   DATA[168,35] := 250.9933;
   DATA[168,36] := 1.681991;
   DATA[168,37] := 189.6789;
   DATA[168,38] := 0.000128152;
   DATA[168,39] := 1.0;
   DATA[169,0] := 2.625628;
   DATA[169,1] := 525.4767;
   DATA[169,2] := 2.0;
   DATA[169,3] := 2.0;
   DATA[169,4] := 262.0802;
   DATA[169,5] := 8.39163;
   DATA[169,6] := 328.2748;
   DATA[169,7] := 2.445904;
   DATA[169,8] := 2.0;
   DATA[169,9] := 2.0;
   DATA[169,10] := 2.0;
   DATA[169,11] := 19.7964;
   DATA[169,12] := 2.209525;
   DATA[169,13] := 963.2146;
   DATA[169,14] := 1.0;
   DATA[169,15] := 2.0;
   DATA[169,16] := 1.0;
   DATA[169,17] := 1.0;
   DATA[169,18] := 1.0;
   DATA[169,19] := 2.0;
   DATA[169,20] := 148.808;
   DATA[169,21] := 156.1138;
   DATA[169,22] := 1.717489;
   DATA[169,23] := 954.14;
   DATA[169,24] := 2.0;
   DATA[169,25] := 2.0;
   DATA[169,26] := 7.875737;
   DATA[169,27] := 145.1423;
   DATA[169,28] := 264.2271;
   DATA[169,29] := 12.26609;
   DATA[169,30] := 1.726737;
   DATA[169,31] := 1.318816;
   DATA[169,32] := 0.7360369;
   DATA[169,33] := 0.3086186;
   DATA[169,34] := 2.0;
   DATA[169,35] := 250.9933;
   DATA[169,36] := 1.681991;
   DATA[169,37] := 189.6789;
   DATA[169,38] := 0.000128152;
   DATA[169,39] := 1.0;
   DATA[170,0] := 2.624027;
   DATA[170,1] := 525.7122;
   DATA[170,2] := 2.0;
   DATA[170,3] := 2.0;
   DATA[170,4] := 262.0802;
   DATA[170,5] := 8.39163;
   DATA[170,6] := 328.2748;
   DATA[170,7] := 2.444366;
   DATA[170,8] := 2.0;
   DATA[170,9] := 2.0;
   DATA[170,10] := 2.0;
   DATA[170,11] := 19.68756;
   DATA[170,12] := 2.210806;
   DATA[170,13] := 963.1745;
   DATA[170,14] := 1.0;
   DATA[170,15] := 2.0;
   DATA[170,16] := 1.0;
   DATA[170,17] := 1.0;
   DATA[170,18] := 1.0;
   DATA[170,19] := 2.0;
   DATA[170,20] := 148.808;
   DATA[170,21] := 156.1138;
   DATA[170,22] := 1.717489;
   DATA[170,23] := 954.1784;
   DATA[170,24] := 2.0;
   DATA[170,25] := 2.0;
   DATA[170,26] := 7.875737;
   DATA[170,27] := 145.1423;
   DATA[170,28] := 264.2271;
   DATA[170,29] := 12.26609;
   DATA[170,30] := 1.726737;
   DATA[170,31] := 1.322019;
   DATA[170,32] := 0.7360369;
   DATA[170,33] := 0.3084265;
   DATA[170,34] := 2.0;
   DATA[170,35] := 250.9933;
   DATA[170,36] := 1.681991;
   DATA[170,37] := 189.6789;
   DATA[170,38] := 0.000128152;
   DATA[170,39] := 1.0;
   DATA[171,0] := 2.612177;
   DATA[171,1] := 525.8692;
   DATA[171,2] := 2.0;
   DATA[171,3] := 2.0;
   DATA[171,4] := 262.0802;
   DATA[171,5] := 8.39163;
   DATA[171,6] := 328.2748;
   DATA[171,7] := 2.443725;
   DATA[171,8] := 2.0;
   DATA[171,9] := 2.0;
   DATA[171,10] := 2.0;
   DATA[171,11] := 19.68756;
   DATA[171,12] := 2.212728;
   DATA[171,13] := 963.3347;
   DATA[171,14] := 1.0;
   DATA[171,15] := 2.0;
   DATA[171,16] := 1.0;
   DATA[171,17] := 1.0;
   DATA[171,18] := 1.0;
   DATA[171,19] := 2.0;
   DATA[171,20] := 148.808;
   DATA[171,21] := 156.1138;
   DATA[171,22] := 1.717489;
   DATA[171,23] := 954.14;
   DATA[171,24] := 2.0;
   DATA[171,25] := 2.0;
   DATA[171,26] := 7.875737;
   DATA[171,27] := 145.1423;
   DATA[171,28] := 264.2271;
   DATA[171,29] := 12.26609;
   DATA[171,30] := 1.726737;
   DATA[171,31] := 1.322019;
   DATA[171,32] := 0.7353967;
   DATA[171,33] := 0.3074016;
   DATA[171,34] := 2.0;
   DATA[171,35] := 250.9933;
   DATA[171,36] := 1.681991;
   DATA[171,37] := 189.6789;
   DATA[171,38] := 0.000128152;
   DATA[171,39] := 1.0;
   DATA[172,0] := 2.59232;
   DATA[172,1] := 526.1832;
   DATA[172,2] := 2.0;
   DATA[172,3] := 2.0;
   DATA[172,4] := 262.0802;
   DATA[172,5] := 8.396116;
   DATA[172,6] := 328.2748;
   DATA[172,7] := 2.441034;
   DATA[172,8] := 2.0;
   DATA[172,9] := 2.0;
   DATA[172,10] := 2.0;
   DATA[172,11] := 19.68756;
   DATA[172,12] := 2.212728;
   DATA[172,13] := 963.6151;
   DATA[172,14] := 1.0;
   DATA[172,15] := 2.0;
   DATA[172,16] := 1.0;
   DATA[172,17] := 1.0;
   DATA[172,18] := 1.0;
   DATA[172,19] := 2.0;
   DATA[172,20] := 148.808;
   DATA[172,21] := 156.1138;
   DATA[172,22] := 1.717489;
   DATA[172,23] := 954.0246;
   DATA[172,24] := 2.0;
   DATA[172,25] := 2.0;
   DATA[172,26] := 7.875737;
   DATA[172,27] := 145.1423;
   DATA[172,28] := 264.2271;
   DATA[172,29] := 12.26609;
   DATA[172,30] := 1.726737;
   DATA[172,31] := 1.302421;
   DATA[172,32] := 0.7352687;
   DATA[172,33] := 0.3070813;
   DATA[172,34] := 2.0;
   DATA[172,35] := 250.9933;
   DATA[172,36] := 1.681991;
   DATA[172,37] := 189.6789;
   DATA[172,38] := 0.000128152;
   DATA[172,39] := 1.0;
   DATA[173,0] := 2.575665;
   DATA[173,1] := 526.3795;
   DATA[173,2] := 2.0;
   DATA[173,3] := 2.0;
   DATA[173,4] := 262.0802;
   DATA[173,5] := 8.396116;
   DATA[173,6] := 328.2748;
   DATA[173,7] := 2.440778;
   DATA[173,8] := 2.0;
   DATA[173,9] := 2.0;
   DATA[173,10] := 2.0;
   DATA[173,11] := 19.68756;
   DATA[173,12] := 2.212728;
   DATA[173,13] := 963.3748;
   DATA[173,14] := 1.0;
   DATA[173,15] := 2.0;
   DATA[173,16] := 1.0;
   DATA[173,17] := 1.0;
   DATA[173,18] := 1.0;
   DATA[173,19] := 2.0;
   DATA[173,20] := 148.808;
   DATA[173,21] := 156.1138;
   DATA[173,22] := 1.717489;
   DATA[173,23] := 954.1015;
   DATA[173,24] := 2.0;
   DATA[173,25] := 2.0;
   DATA[173,26] := 7.875737;
   DATA[173,27] := 145.1423;
   DATA[173,28] := 264.2271;
   DATA[173,29] := 12.26609;
   DATA[173,30] := 1.725583;
   DATA[173,31] := 1.292046;
   DATA[173,32] := 0.7352687;
   DATA[173,33] := 0.3070813;
   DATA[173,34] := 2.0;
   DATA[173,35] := 250.8812;
   DATA[173,36] := 1.681991;
   DATA[173,37] := 189.6789;
   DATA[173,38] := 0.000128152;
   DATA[173,39] := 1.0;
   DATA[174,0] := 2.554527;
   DATA[174,1] := 526.615;
   DATA[174,2] := 2.0;
   DATA[174,3] := 2.0;
   DATA[174,4] := 262.0802;
   DATA[174,5] := 8.396116;
   DATA[174,6] := 328.2748;
   DATA[174,7] := 2.440778;
   DATA[174,8] := 2.0;
   DATA[174,9] := 2.0;
   DATA[174,10] := 2.0;
   DATA[174,11] := 19.68756;
   DATA[174,12] := 2.211831;
   DATA[174,13] := 963.7353;
   DATA[174,14] := 1.0;
   DATA[174,15] := 2.0;
   DATA[174,16] := 1.0;
   DATA[174,17] := 1.0;
   DATA[174,18] := 1.0;
   DATA[174,19] := 2.0;
   DATA[174,20] := 148.808;
   DATA[174,21] := 156.1138;
   DATA[174,22] := 1.717489;
   DATA[174,23] := 954.5245;
   DATA[174,24] := 2.0;
   DATA[174,25] := 2.0;
   DATA[174,26] := 7.875737;
   DATA[174,27] := 145.1423;
   DATA[174,28] := 264.2271;
   DATA[174,29] := 12.26609;
   DATA[174,30] := 1.725455;
   DATA[174,31] := 1.290893;
   DATA[174,32] := 0.7352687;
   DATA[174,33] := 0.3065048;
   DATA[174,34] := 2.0;
   DATA[174,35] := 250.8812;
   DATA[174,36] := 1.681991;
   DATA[174,37] := 189.6469;
   DATA[174,38] := 0.000128152;
   DATA[174,39] := 1.0;
   DATA[175,0] := 2.535951;
   DATA[175,1] := 526.5757;
   DATA[175,2] := 2.0;
   DATA[175,3] := 2.0;
   DATA[175,4] := 262.0802;
   DATA[175,5] := 8.396116;
   DATA[175,6] := 328.2748;
   DATA[175,7] := 2.441547;
   DATA[175,8] := 2.0;
   DATA[175,9] := 2.0;
   DATA[175,10] := 2.0;
   DATA[175,11] := 19.68756;
   DATA[175,12] := 2.210294;
   DATA[175,13] := 963.7353;
   DATA[175,14] := 1.0;
   DATA[175,15] := 2.0;
   DATA[175,16] := 1.0;
   DATA[175,17] := 1.0;
   DATA[175,18] := 1.0;
   DATA[175,19] := 2.0;
   DATA[175,20] := 148.808;
   DATA[175,21] := 156.1138;
   DATA[175,22] := 1.717489;
   DATA[175,23] := 955.1013;
   DATA[175,24] := 2.0;
   DATA[175,25] := 2.0;
   DATA[175,26] := 7.875737;
   DATA[175,27] := 145.1423;
   DATA[175,28] := 264.2271;
   DATA[175,29] := 12.11228;
   DATA[175,30] := 1.725455;
   DATA[175,31] := 1.285001;
   DATA[175,32] := 0.7352687;
   DATA[175,33] := 0.3065048;
   DATA[175,34] := 2.0;
   DATA[175,35] := 250.8812;
   DATA[175,36] := 1.681991;
   DATA[175,37] := 189.5347;
   DATA[175,38] := 0.000128152;
   DATA[175,39] := 1.0;
   DATA[176,0] := 2.520257;
   DATA[176,1] := 526.6542;
   DATA[176,2] := 2.0;
   DATA[176,3] := 2.0;
   DATA[176,4] := 262.0802;
   DATA[176,5] := 8.396116;
   DATA[176,6] := 328.2748;
   DATA[176,7] := 2.443597;
   DATA[176,8] := 2.0;
   DATA[176,9] := 2.0;
   DATA[176,10] := 2.0;
   DATA[176,11] := 19.68756;
   DATA[176,12] := 2.210166;
   DATA[176,13] := 963.535;
   DATA[176,14] := 1.0;
   DATA[176,15] := 2.0;
   DATA[176,16] := 1.0;
   DATA[176,17] := 1.0;
   DATA[176,18] := 1.0;
   DATA[176,19] := 2.0;
   DATA[176,20] := 148.808;
   DATA[176,21] := 156.0369;
   DATA[176,22] := 1.717489;
   DATA[176,23] := 955.3704;
   DATA[176,24] := 2.0;
   DATA[176,25] := 2.0;
   DATA[176,26] := 7.875737;
   DATA[176,27] := 145.1423;
   DATA[176,28] := 264.2271;
   DATA[176,29] := 12.11228;
   DATA[176,30] := 1.725455;
   DATA[176,31] := 1.272704;
   DATA[176,32] := 0.7352687;
   DATA[176,33] := 0.3065048;
   DATA[176,34] := 2.0;
   DATA[176,35] := 250.8812;
   DATA[176,36] := 1.681991;
   DATA[176,37] := 189.5347;
   DATA[176,38] := 0.000128152;
   DATA[176,39] := 1.0;
   DATA[177,0] := 2.501041;
   DATA[177,1] := 526.8113;
   DATA[177,2] := 2.0;
   DATA[177,3] := 2.0;
   DATA[177,4] := 262.0802;
   DATA[177,5] := 8.396116;
   DATA[177,6] := 328.2748;
   DATA[177,7] := 2.445391;
   DATA[177,8] := 2.0;
   DATA[177,9] := 2.0;
   DATA[177,10] := 2.0;
   DATA[177,11] := 19.71957;
   DATA[177,12] := 2.210934;
   DATA[177,13] := 963.6151;
   DATA[177,14] := 1.0;
   DATA[177,15] := 2.0;
   DATA[177,16] := 1.0;
   DATA[177,17] := 1.0;
   DATA[177,18] := 1.0;
   DATA[177,19] := 2.0;
   DATA[177,20] := 148.808;
   DATA[177,21] := 155.9087;
   DATA[177,22] := 1.717489;
   DATA[177,23] := 955.2935;
   DATA[177,24] := 2.0;
   DATA[177,25] := 2.0;
   DATA[177,26] := 7.875737;
   DATA[177,27] := 145.091;
   DATA[177,28] := 264.2271;
   DATA[177,29] := 12.11228;
   DATA[177,30] := 1.725455;
   DATA[177,31] := 1.272064;
   DATA[177,32] := 0.7352687;
   DATA[177,33] := 0.3065048;
   DATA[177,34] := 2.0;
   DATA[177,35] := 250.8812;
   DATA[177,36] := 1.681991;
   DATA[177,37] := 189.5347;
   DATA[177,38] := 0.000128152;
   DATA[177,39] := 1.0;
   DATA[178,0] := 2.48823;
   DATA[178,1] := 527.2038;
   DATA[178,2] := 2.0;
   DATA[178,3] := 2.0;
   DATA[178,4] := 262.0802;
   DATA[178,5] := 8.396116;
   DATA[178,6] := 328.2748;
   DATA[178,7] := 2.445391;
   DATA[178,8] := 2.0;
   DATA[178,9] := 2.0;
   DATA[178,10] := 2.0;
   DATA[178,11] := 19.74198;
   DATA[178,12] := 2.213368;
   DATA[178,13] := 963.9756;
   DATA[178,14] := 1.0;
   DATA[178,15] := 2.0;
   DATA[178,16] := 1.0;
   DATA[178,17] := 1.0;
   DATA[178,18] := 1.0;
   DATA[178,19] := 2.0;
   DATA[178,20] := 148.808;
   DATA[178,21] := 155.9087;
   DATA[178,22] := 1.717361;
   DATA[178,23] := 956.0626;
   DATA[178,24] := 2.0;
   DATA[178,25] := 2.0;
   DATA[178,26] := 7.875737;
   DATA[178,27] := 145.091;
   DATA[178,28] := 264.2271;
   DATA[178,29] := 12.11228;
   DATA[178,30] := 1.725455;
   DATA[178,31] := 1.273216;
   DATA[178,32] := 0.7352687;
   DATA[178,33] := 0.3084265;
   DATA[178,34] := 2.0;
   DATA[178,35] := 250.8812;
   DATA[178,36] := 1.681991;
   DATA[178,37] := 189.5347;
   DATA[178,38] := 0.000128152;
   DATA[178,39] := 1.0;
   DATA[179,0] := 2.468693;
   DATA[179,1] := 527.1646;
   DATA[179,2] := 2.0;
   DATA[179,3] := 2.0;
   DATA[179,4] := 262.0802;
   DATA[179,5] := 8.396116;
   DATA[179,6] := 328.2748;
   DATA[179,7] := 2.445391;
   DATA[179,8] := 2.0;
   DATA[179,9] := 2.0;
   DATA[179,10] := 2.0;
   DATA[179,11] := 19.74198;
   DATA[179,12] := 2.213368;
   DATA[179,13] := 964.4562;
   DATA[179,14] := 1.0;
   DATA[179,15] := 2.0;
   DATA[179,16] := 1.0;
   DATA[179,17] := 1.0;
   DATA[179,18] := 1.0;
   DATA[179,19] := 2.0;
   DATA[179,20] := 148.808;
   DATA[179,21] := 155.9087;
   DATA[179,22] := 1.716208;
   DATA[179,23] := 956.3317;
   DATA[179,24] := 2.0;
   DATA[179,25] := 2.0;
   DATA[179,26] := 7.875737;
   DATA[179,27] := 144.9116;
   DATA[179,28] := 264.2271;
   DATA[179,29] := 12.11228;
   DATA[179,30] := 1.725455;
   DATA[179,31] := 1.281542;
   DATA[179,32] := 0.7352687;
   DATA[179,33] := 0.3084265;
   DATA[179,34] := 2.0;
   DATA[179,35] := 250.8812;
   DATA[179,36] := 1.681991;
   DATA[179,37] := 189.5668;
   DATA[179,38] := 0.000128152;
   DATA[179,39] := 1.0;
   DATA[180,0] := 2.451078;
   DATA[180,1] := 527.5571;
   DATA[180,2] := 2.0;
   DATA[180,3] := 2.0;
   DATA[180,4] := 262.0802;
   DATA[180,5] := 8.395475;
   DATA[180,6] := 328.2748;
   DATA[180,7] := 2.445391;
   DATA[180,8] := 2.0;
   DATA[180,9] := 2.0;
   DATA[180,10] := 2.0;
   DATA[180,11] := 19.74198;
   DATA[180,12] := 2.213368;
   DATA[180,13] := 964.8568;
   DATA[180,14] := 1.0;
   DATA[180,15] := 2.0;
   DATA[180,16] := 1.0;
   DATA[180,17] := 1.0;
   DATA[180,18] := 1.0;
   DATA[180,19] := 2.0;
   DATA[180,20] := 148.808;
   DATA[180,21] := 155.9856;
   DATA[180,22] := 1.716208;
   DATA[180,23] := 956.4855;
   DATA[180,24] := 2.0;
   DATA[180,25] := 2.0;
   DATA[180,26] := 7.875737;
   DATA[180,27] := 144.9116;
   DATA[180,28] := 264.2271;
   DATA[180,29] := 12.11228;
   DATA[180,30] := 1.726993;
   DATA[180,31] := 1.281542;
   DATA[180,32] := 0.7352687;
   DATA[180,33] := 0.3084265;
   DATA[180,34] := 2.0;
   DATA[180,35] := 250.8812;
   DATA[180,36] := 1.681991;
   DATA[180,37] := 189.759;
   DATA[180,38] := 0.000128152;
   DATA[180,39] := 1.0;
   DATA[181,0] := 2.440188;
   DATA[181,1] := 527.8318;
   DATA[181,2] := 2.0;
   DATA[181,3] := 2.0;
   DATA[181,4] := 262.0802;
   DATA[181,5] := 8.395475;
   DATA[181,6] := 328.2748;
   DATA[181,7] := 2.44411;
   DATA[181,8] := 2.0;
   DATA[181,9] := 2.0;
   DATA[181,10] := 2.0;
   DATA[181,11] := 19.72598;
   DATA[181,12] := 2.213368;
   DATA[181,13] := 965.2573;
   DATA[181,14] := 1.0;
   DATA[181,15] := 2.0;
   DATA[181,16] := 1.0;
   DATA[181,17] := 1.0;
   DATA[181,18] := 1.0;
   DATA[181,19] := 2.0;
   DATA[181,20] := 148.808;
   DATA[181,21] := 156.0625;
   DATA[181,22] := 1.71813;
   DATA[181,23] := 957.2161;
   DATA[181,24] := 2.0;
   DATA[181,25] := 2.0;
   DATA[181,26] := 7.875737;
   DATA[181,27] := 144.9116;
   DATA[181,28] := 264.2271;
   DATA[181,29] := 12.11228;
   DATA[181,30] := 1.726993;
   DATA[181,31] := 1.281542;
   DATA[181,32] := 0.7352687;
   DATA[181,33] := 0.3084265;
   DATA[181,34] := 2.0;
   DATA[181,35] := 250.9933;
   DATA[181,36] := 1.681991;
   DATA[181,37] := 189.759;
   DATA[181,38] := 0.000128152;
   DATA[181,39] := 1.0;
   DATA[182,0] := 2.429619;
   DATA[182,1] := 527.8318;
   DATA[182,2] := 2.0;
   DATA[182,3] := 2.0;
   DATA[182,4] := 262.0802;
   DATA[182,5] := 8.395475;
   DATA[182,6] := 328.2748;
   DATA[182,7] := 2.44411;
   DATA[182,8] := 2.0;
   DATA[182,9] := 2.0;
   DATA[182,10] := 2.0;
   DATA[182,11] := 19.72598;
   DATA[182,12] := 2.214137;
   DATA[182,13] := 965.5778;
   DATA[182,14] := 1.0;
   DATA[182,15] := 2.0;
   DATA[182,16] := 1.0;
   DATA[182,17] := 1.0;
   DATA[182,18] := 1.0;
   DATA[182,19] := 2.0;
   DATA[182,20] := 148.808;
   DATA[182,21] := 156.0625;
   DATA[182,22] := 1.718771;
   DATA[182,23] := 957.0623;
   DATA[182,24] := 2.0;
   DATA[182,25] := 2.0;
   DATA[182,26] := 7.875737;
   DATA[182,27] := 144.9116;
   DATA[182,28] := 264.131;
   DATA[182,29] := 12.11228;
   DATA[182,30] := 1.728659;
   DATA[182,31] := 1.281542;
   DATA[182,32] := 0.7352687;
   DATA[182,33] := 0.3084265;
   DATA[182,34] := 2.0;
   DATA[182,35] := 251.1215;
   DATA[182,36] := 1.681991;
   DATA[182,37] := 189.759;
   DATA[182,38] := 0.000128152;
   DATA[182,39] := 1.0;
   DATA[183,0] := 2.426737;
   DATA[183,1] := 528.3421;
   DATA[183,2] := 2.0;
   DATA[183,3] := 2.0;
   DATA[183,4] := 262.0802;
   DATA[183,5] := 8.395475;
   DATA[183,6] := 328.2748;
   DATA[183,7] := 2.44411;
   DATA[183,8] := 2.0;
   DATA[183,9] := 2.0;
   DATA[183,10] := 2.0;
   DATA[183,11] := 19.72598;
   DATA[183,12] := 2.214137;
   DATA[183,13] := 965.778;
   DATA[183,14] := 1.0;
   DATA[183,15] := 2.0;
   DATA[183,16] := 1.0;
   DATA[183,17] := 1.0;
   DATA[183,18] := 1.0;
   DATA[183,19] := 2.0;
   DATA[183,20] := 148.808;
   DATA[183,21] := 156.0625;
   DATA[183,22] := 1.718771;
   DATA[183,23] := 957.5621;
   DATA[183,24] := 2.0;
   DATA[183,25] := 2.0;
   DATA[183,26] := 7.875737;
   DATA[183,27] := 144.9116;
   DATA[183,28] := 264.131;
   DATA[183,29] := 12.11228;
   DATA[183,30] := 1.728916;
   DATA[183,31] := 1.275138;
   DATA[183,32] := 0.7352687;
   DATA[183,33] := 0.3084265;
   DATA[183,34] := 2.0;
   DATA[183,35] := 251.1215;
   DATA[183,36] := 1.681991;
   DATA[183,37] := 189.759;
   DATA[183,38] := 0.000128152;
   DATA[183,39] := 1.0;
   DATA[184,0] := 2.428018;
   DATA[184,1] := 528.2636;
   DATA[184,2] := 2.0;
   DATA[184,3] := 2.0;
   DATA[184,4] := 262.0802;
   DATA[184,5] := 8.393232;
   DATA[184,6] := 328.2748;
   DATA[184,7] := 2.443469;
   DATA[184,8] := 2.0;
   DATA[184,9] := 2.0;
   DATA[184,10] := 2.0;
   DATA[184,11] := 19.74838;
   DATA[184,12] := 2.211575;
   DATA[184,13] := 965.6178;
   DATA[184,14] := 1.0;
   DATA[184,15] := 2.0;
   DATA[184,16] := 1.0;
   DATA[184,17] := 1.0;
   DATA[184,18] := 1.0;
   DATA[184,19] := 2.0;
   DATA[184,20] := 148.808;
   DATA[184,21] := 156.0625;
   DATA[184,22] := 1.718771;
   DATA[184,23] := 957.6775;
   DATA[184,24] := 2.0;
   DATA[184,25] := 2.0;
   DATA[184,26] := 7.875737;
   DATA[184,27] := 144.9116;
   DATA[184,28] := 264.131;
   DATA[184,29] := 12.11228;
   DATA[184,30] := 1.729172;
   DATA[184,31] := 1.288331;
   DATA[184,32] := 0.7352687;
   DATA[184,33] := 0.3068891;
   DATA[184,34] := 2.0;
   DATA[184,35] := 251.1215;
   DATA[184,36] := 1.681991;
   DATA[184,37] := 189.9032;
   DATA[184,38] := 0.000128152;
   DATA[184,39] := 1.0;
   DATA[185,0] := 2.480863;
   DATA[185,1] := 528.2244;
   DATA[185,2] := 2.0;
   DATA[185,3] := 2.0;
   DATA[185,4] := 262.0802;
   DATA[185,5] := 8.393232;
   DATA[185,6] := 328.2748;
   DATA[185,7] := 2.442188;
   DATA[185,8] := 2.0;
   DATA[185,9] := 2.0;
   DATA[185,10] := 2.0;
   DATA[185,11] := 19.77079;
   DATA[185,12] := 2.210166;
   DATA[185,13] := 965.9382;
   DATA[185,14] := 1.0;
   DATA[185,15] := 2.0;
   DATA[185,16] := 1.0;
   DATA[185,17] := 1.0;
   DATA[185,18] := 1.0;
   DATA[185,19] := 2.0;
   DATA[185,20] := 148.808;
   DATA[185,21] := 156.0625;
   DATA[185,22] := 1.717489;
   DATA[185,23] := 957.7928;
   DATA[185,24] := 2.0;
   DATA[185,25] := 2.0;
   DATA[185,26] := 7.875737;
   DATA[185,27] := 144.7065;
   DATA[185,28] := 264.131;
   DATA[185,29] := 12.11228;
   DATA[185,30] := 1.729172;
   DATA[185,31] := 1.291149;
   DATA[185,32] := 0.7353967;
   DATA[185,33] := 0.3072094;
   DATA[185,34] := 2.0;
   DATA[185,35] := 251.2657;
   DATA[185,36] := 1.681991;
   DATA[185,37] := 189.9032;
   DATA[185,38] := 0.000128152;
   DATA[185,39] := 1.0;
   DATA[186,0] := 2.528264;
   DATA[186,1] := 528.0674;
   DATA[186,2] := 2.0;
   DATA[186,3] := 2.0;
   DATA[186,4] := 262.0802;
   DATA[186,5] := 8.393232;
   DATA[186,6] := 328.2748;
   DATA[186,7] := 2.442188;
   DATA[186,8] := 2.0;
   DATA[186,9] := 2.0;
   DATA[186,10] := 2.0;
   DATA[186,11] := 19.77079;
   DATA[186,12] := 2.210166;
   DATA[186,13] := 965.8582;
   DATA[186,14] := 1.0;
   DATA[186,15] := 2.0;
   DATA[186,16] := 1.0;
   DATA[186,17] := 1.0;
   DATA[186,18] := 1.0;
   DATA[186,19] := 2.0;
   DATA[186,20] := 148.808;
   DATA[186,21] := 156.0625;
   DATA[186,22] := 1.717489;
   DATA[186,23] := 957.8313;
   DATA[186,24] := 2.0;
   DATA[186,25] := 2.0;
   DATA[186,26] := 7.875737;
   DATA[186,27] := 144.7065;
   DATA[186,28] := 264.131;
   DATA[186,29] := 12.11228;
   DATA[186,30] := 1.729172;
   DATA[186,31] := 1.281798;
   DATA[186,32] := 0.7353967;
   DATA[186,33] := 0.3072094;
   DATA[186,34] := 2.0;
   DATA[186,35] := 251.2657;
   DATA[186,36] := 1.681991;
   DATA[186,37] := 189.9032;
   DATA[186,38] := 0.000128152;
   DATA[186,39] := 1.0;
   DATA[187,0] := 2.56958;
   DATA[187,1] := 528.0674;
   DATA[187,2] := 2.0;
   DATA[187,3] := 2.0;
   DATA[187,4] := 262.0802;
   DATA[187,5] := 8.393232;
   DATA[187,6] := 328.2748;
   DATA[187,7] := 2.441034;
   DATA[187,8] := 2.0;
   DATA[187,9] := 2.0;
   DATA[187,10] := 2.0;
   DATA[187,11] := 19.73878;
   DATA[187,12] := 2.210166;
   DATA[187,13] := 965.5778;
   DATA[187,14] := 1.0;
   DATA[187,15] := 2.0;
   DATA[187,16] := 1.0;
   DATA[187,17] := 1.0;
   DATA[187,18] := 1.0;
   DATA[187,19] := 2.0;
   DATA[187,20] := 148.808;
   DATA[187,21] := 156.0625;
   DATA[187,22] := 1.717489;
   DATA[187,23] := 958.2543;
   DATA[187,24] := 2.0;
   DATA[187,25] := 2.0;
   DATA[187,26] := 7.875737;
   DATA[187,27] := 144.7065;
   DATA[187,28] := 264.131;
   DATA[187,29] := 12.11228;
   DATA[187,30] := 1.729172;
   DATA[187,31] := 1.281286;
   DATA[187,32] := 0.7353967;
   DATA[187,33] := 0.3072094;
   DATA[187,34] := 2.0;
   DATA[187,35] := 251.2657;
   DATA[187,36] := 1.681991;
   DATA[187,37] := 189.9032;
   DATA[187,38] := 0.000128152;
   DATA[187,39] := 1.0;
   DATA[188,0] := 2.601287;
   DATA[188,1] := 528.3421;
   DATA[188,2] := 2.0;
   DATA[188,3] := 2.0;
   DATA[188,4] := 262.0802;
   DATA[188,5] := 8.393232;
   DATA[188,6] := 328.2748;
   DATA[188,7] := 2.440521;
   DATA[188,8] := 2.0;
   DATA[188,9] := 2.0;
   DATA[188,10] := 2.0;
   DATA[188,11] := 19.70037;
   DATA[188,12] := 2.212984;
   DATA[188,13] := 965.4576;
   DATA[188,14] := 1.0;
   DATA[188,15] := 2.0;
   DATA[188,16] := 1.0;
   DATA[188,17] := 1.0;
   DATA[188,18] := 1.0;
   DATA[188,19] := 2.0;
   DATA[188,20] := 148.808;
   DATA[188,21] := 156.0625;
   DATA[188,22] := 1.717489;
   DATA[188,23] := 958.3312;
   DATA[188,24] := 2.0;
   DATA[188,25] := 2.0;
   DATA[188,26] := 7.876378;
   DATA[188,27] := 144.7065;
   DATA[188,28] := 264.131;
   DATA[188,29] := 12.11228;
   DATA[188,30] := 1.729172;
   DATA[188,31] := 1.273216;
   DATA[188,32] := 0.7353967;
   DATA[188,33] := 0.3072094;
   DATA[188,34] := 2.0;
   DATA[188,35] := 251.2657;
   DATA[188,36] := 1.681991;
   DATA[188,37] := 189.9032;
   DATA[188,38] := 0.000128152;
   DATA[188,39] := 1.0;
   DATA[189,0] := 2.644525;
   DATA[189,1] := 528.4207;
   DATA[189,2] := 2.0;
   DATA[189,3] := 2.0;
   DATA[189,4] := 262.0802;
   DATA[189,5] := 8.391951;
   DATA[189,6] := 328.2748;
   DATA[189,7] := 2.440521;
   DATA[189,8] := 2.0;
   DATA[189,9] := 2.0;
   DATA[189,10] := 2.0;
   DATA[189,11] := 19.65875;
   DATA[189,12] := 2.212984;
   DATA[189,13] := 965.3375;
   DATA[189,14] := 1.0;
   DATA[189,15] := 2.0;
   DATA[189,16] := 1.0;
   DATA[189,17] := 1.0;
   DATA[189,18] := 1.0;
   DATA[189,19] := 2.0;
   DATA[189,20] := 148.808;
   DATA[189,21] := 156.0625;
   DATA[189,22] := 1.717489;
   DATA[189,23] := 958.5234;
   DATA[189,24] := 2.0;
   DATA[189,25] := 2.0;
   DATA[189,26] := 7.878621;
   DATA[189,27] := 144.7065;
   DATA[189,28] := 264.131;
   DATA[189,29] := 12.26609;
   DATA[189,30] := 1.729172;
   DATA[189,31] := 1.271935;
   DATA[189,32] := 0.7353967;
   DATA[189,33] := 0.3072094;
   DATA[189,34] := 2.0;
   DATA[189,35] := 251.2657;
   DATA[189,36] := 1.681991;
   DATA[189,37] := 189.9032;
   DATA[189,38] := 0.000128152;
   DATA[189,39] := 1.0;
   DATA[190,0] := 2.665663;
   DATA[190,1] := 528.1851;
   DATA[190,2] := 2.0;
   DATA[190,3] := 2.0;
   DATA[190,4] := 262.0802;
   DATA[190,5] := 8.391951;
   DATA[190,6] := 328.2748;
   DATA[190,7] := 2.440521;
   DATA[190,8] := 2.0;
   DATA[190,9] := 2.0;
   DATA[190,10] := 2.0;
   DATA[190,11] := 19.64274;
   DATA[190,12] := 2.212984;
   DATA[190,13] := 965.3375;
   DATA[190,14] := 1.0;
   DATA[190,15] := 2.0;
   DATA[190,16] := 1.0;
   DATA[190,17] := 1.0;
   DATA[190,18] := 1.0;
   DATA[190,19] := 2.0;
   DATA[190,20] := 148.808;
   DATA[190,21] := 156.0625;
   DATA[190,22] := 1.717489;
   DATA[190,23] := 959.0618;
   DATA[190,24] := 2.0;
   DATA[190,25] := 2.0;
   DATA[190,26] := 7.878621;
   DATA[190,27] := 144.7065;
   DATA[190,28] := 264.131;
   DATA[190,29] := 12.26609;
   DATA[190,30] := 1.729172;
   DATA[190,31] := 1.271935;
   DATA[190,32] := 0.7353967;
   DATA[190,33] := 0.306761;
   DATA[190,34] := 2.0;
   DATA[190,35] := 251.1055;
   DATA[190,36] := 1.681991;
   DATA[190,37] := 189.9032;
   DATA[190,38] := 0.000128152;
   DATA[190,39] := 1.0;
   DATA[191,0] := 2.670788;
   DATA[191,1] := 527.8711;
   DATA[191,2] := 2.0;
   DATA[191,3] := 2.0;
   DATA[191,4] := 262.0802;
   DATA[191,5] := 8.391951;
   DATA[191,6] := 328.2748;
   DATA[191,7] := 2.440521;
   DATA[191,8] := 2.0;
   DATA[191,9] := 2.0;
   DATA[191,10] := 2.0;
   DATA[191,11] := 19.64274;
   DATA[191,12] := 2.212984;
   DATA[191,13] := 965.3775;
   DATA[191,14] := 1.0;
   DATA[191,15] := 2.0;
   DATA[191,16] := 1.0;
   DATA[191,17] := 1.0;
   DATA[191,18] := 1.0;
   DATA[191,19] := 2.0;
   DATA[191,20] := 148.808;
   DATA[191,21] := 156.0625;
   DATA[191,22] := 1.717489;
   DATA[191,23] := 958.9849;
   DATA[191,24] := 2.0;
   DATA[191,25] := 2.0;
   DATA[191,26] := 7.878621;
   DATA[191,27] := 144.7065;
   DATA[191,28] := 264.131;
   DATA[191,29] := 12.26609;
   DATA[191,30] := 1.729172;
   DATA[191,31] := 1.281542;
   DATA[191,32] := 0.7353967;
   DATA[191,33] := 0.3065048;
   DATA[191,34] := 2.0;
   DATA[191,35] := 251.1055;
   DATA[191,36] := 1.681991;
   DATA[191,37] := 189.9032;
   DATA[191,38] := 0.000128152;
   DATA[191,39] := 1.0;
   DATA[192,0] := 2.656055;
   DATA[192,1] := 528.1459;
   DATA[192,2] := 2.0;
   DATA[192,3] := 2.0;
   DATA[192,4] := 262.0802;
   DATA[192,5] := 8.391951;
   DATA[192,6] := 328.2748;
   DATA[192,7] := 2.440521;
   DATA[192,8] := 2.0;
   DATA[192,9] := 2.0;
   DATA[192,10] := 2.0;
   DATA[192,11] := 19.64274;
   DATA[192,12] := 2.213624;
   DATA[192,13] := 965.1772;
   DATA[192,14] := 1.0;
   DATA[192,15] := 2.0;
   DATA[192,16] := 1.0;
   DATA[192,17] := 1.0;
   DATA[192,18] := 1.0;
   DATA[192,19] := 2.0;
   DATA[192,20] := 148.808;
   DATA[192,21] := 156.0625;
   DATA[192,22] := 1.717489;
   DATA[192,23] := 958.9464;
   DATA[192,24] := 2.0;
   DATA[192,25] := 2.0;
   DATA[192,26] := 7.877019;
   DATA[192,27] := 144.7065;
   DATA[192,28] := 264.131;
   DATA[192,29] := 12.26609;
   DATA[192,30] := 1.729172;
   DATA[192,31] := 1.298578;
   DATA[192,32] := 0.7353967;
   DATA[192,33] := 0.3065048;
   DATA[192,34] := 2.0;
   DATA[192,35] := 251.1055;
   DATA[192,36] := 1.681991;
   DATA[192,37] := 189.9032;
   DATA[192,38] := 0.000128152;
   DATA[192,39] := 1.0;
   DATA[193,0] := 2.633315;
   DATA[193,1] := 527.4001;
   DATA[193,2] := 2.0;
   DATA[193,3] := 2.0;
   DATA[193,4] := 262.0802;
   DATA[193,5] := 8.391951;
   DATA[193,6] := 328.2748;
   DATA[193,7] := 2.442828;
   DATA[193,8] := 2.0;
   DATA[193,9] := 2.0;
   DATA[193,10] := 2.0;
   DATA[193,11] := 19.64274;
   DATA[193,12] := 2.213624;
   DATA[193,13] := 965.1772;
   DATA[193,14] := 1.0;
   DATA[193,15] := 2.0;
   DATA[193,16] := 1.0;
   DATA[193,17] := 1.0;
   DATA[193,18] := 1.0;
   DATA[193,19] := 2.0;
   DATA[193,20] := 148.808;
   DATA[193,21] := 156.0625;
   DATA[193,22] := 1.717489;
   DATA[193,23] := 958.9849;
   DATA[193,24] := 2.0;
   DATA[193,25] := 2.0;
   DATA[193,26] := 7.876378;
   DATA[193,27] := 144.7065;
   DATA[193,28] := 264.131;
   DATA[193,29] := 12.26609;
   DATA[193,30] := 1.729172;
   DATA[193,31] := 1.302037;
   DATA[193,32] := 0.7353967;
   DATA[193,33] := 0.3065048;
   DATA[193,34] := 2.0;
   DATA[193,35] := 251.1055;
   DATA[193,36] := 1.681991;
   DATA[193,37] := 189.9032;
   DATA[193,38] := 0.000128152;
   DATA[193,39] := 1.0;
   DATA[194,0] := 2.624027;
   DATA[194,1] := 527.1646;
   DATA[194,2] := 2.0;
   DATA[194,3] := 2.0;
   DATA[194,4] := 262.0802;
   DATA[194,5] := 8.391951;
   DATA[194,6] := 328.2748;
   DATA[194,7] := 2.442956;
   DATA[194,8] := 2.0;
   DATA[194,9] := 2.0;
   DATA[194,10] := 2.0;
   DATA[194,11] := 19.64274;
   DATA[194,12] := 2.213624;
   DATA[194,13] := 964.9369;
   DATA[194,14] := 1.0;
   DATA[194,15] := 2.0;
   DATA[194,16] := 1.0;
   DATA[194,17] := 1.0;
   DATA[194,18] := 1.0;
   DATA[194,19] := 2.0;
   DATA[194,20] := 148.808;
   DATA[194,21] := 156.0625;
   DATA[194,22] := 1.717489;
   DATA[194,23] := 958.9464;
   DATA[194,24] := 2.0;
   DATA[194,25] := 2.0;
   DATA[194,26] := 7.875737;
   DATA[194,27] := 144.7065;
   DATA[194,28] := 264.131;
   DATA[194,29] := 12.26609;
   DATA[194,30] := 1.728531;
   DATA[194,31] := 1.302293;
   DATA[194,32] := 0.7353967;
   DATA[194,33] := 0.3065048;
   DATA[194,34] := 2.0;
   DATA[194,35] := 251.1055;
   DATA[194,36] := 1.681991;
   DATA[194,37] := 189.9032;
   DATA[194,38] := 0.000128152;
   DATA[194,39] := 1.0;
   DATA[195,0] := 2.623387;
   DATA[195,1] := 527.4001;
   DATA[195,2] := 2.0;
   DATA[195,3] := 2.0;
   DATA[195,4] := 262.0802;
   DATA[195,5] := 8.391951;
   DATA[195,6] := 328.2748;
   DATA[195,7] := 2.44616;
   DATA[195,8] := 2.0;
   DATA[195,9] := 2.0;
   DATA[195,10] := 2.0;
   DATA[195,11] := 19.64274;
   DATA[195,12] := 2.213624;
   DATA[195,13] := 965.0571;
   DATA[195,14] := 1.0;
   DATA[195,15] := 2.0;
   DATA[195,16] := 1.0;
   DATA[195,17] := 1.0;
   DATA[195,18] := 1.0;
   DATA[195,19] := 2.0;
   DATA[195,20] := 148.808;
   DATA[195,21] := 156.0625;
   DATA[195,22] := 1.717489;
   DATA[195,23] := 958.9464;
   DATA[195,24] := 2.0;
   DATA[195,25] := 2.0;
   DATA[195,26] := 7.875737;
   DATA[195,27] := 144.7578;
   DATA[195,28] := 264.131;
   DATA[195,29] := 12.26609;
   DATA[195,30] := 1.72725;
   DATA[195,31] := 1.29307;
   DATA[195,32] := 0.7353967;
   DATA[195,33] := 0.3065048;
   DATA[195,34] := 2.0;
   DATA[195,35] := 251.1055;
   DATA[195,36] := 1.681991;
   DATA[195,37] := 189.8071;
   DATA[195,38] := 0.000128152;
   DATA[195,39] := 1.0;
   DATA[196,0] := 2.617942;
   DATA[196,1] := 527.4786;
   DATA[196,2] := 2.0;
   DATA[196,3] := 2.0;
   DATA[196,4] := 262.0802;
   DATA[196,5] := 8.391951;
   DATA[196,6] := 328.2748;
   DATA[196,7] := 2.44616;
   DATA[196,8] := 2.0;
   DATA[196,9] := 2.0;
   DATA[196,10] := 2.0;
   DATA[196,11] := 19.65875;
   DATA[196,12] := 2.213624;
   DATA[196,13] := 965.1772;
   DATA[196,14] := 1.0;
   DATA[196,15] := 2.0;
   DATA[196,16] := 1.0;
   DATA[196,17] := 1.0;
   DATA[196,18] := 1.0;
   DATA[196,19] := 2.0;
   DATA[196,20] := 148.808;
   DATA[196,21] := 156.0625;
   DATA[196,22] := 1.714029;
   DATA[196,23] := 959.1771;
   DATA[196,24] := 2.0;
   DATA[196,25] := 2.0;
   DATA[196,26] := 7.875737;
   DATA[196,27] := 144.7578;
   DATA[196,28] := 264.131;
   DATA[196,29] := 12.26609;
   DATA[196,30] := 1.726737;
   DATA[196,31] := 1.273345;
   DATA[196,32] := 0.7353967;
   DATA[196,33] := 0.3065048;
   DATA[196,34] := 2.0;
   DATA[196,35] := 250.9773;
   DATA[196,36] := 1.826162;
   DATA[196,37] := 189.6789;
   DATA[196,38] := 0.000128152;
   DATA[196,39] := 1.0;
   DATA[197,0] := 2.596163;
   DATA[197,1] := 527.2038;
   DATA[197,2] := 2.0;
   DATA[197,3] := 2.0;
   DATA[197,4] := 262.0802;
   DATA[197,5] := 8.391951;
   DATA[197,6] := 328.2748;
   DATA[197,7] := 2.443982;
   DATA[197,8] := 2.0;
   DATA[197,9] := 2.0;
   DATA[197,10] := 2.0;
   DATA[197,11] := 19.67155;
   DATA[197,12] := 2.213624;
   DATA[197,13] := 964.9369;
   DATA[197,14] := 1.0;
   DATA[197,15] := 2.0;
   DATA[197,16] := 1.0;
   DATA[197,17] := 1.0;
   DATA[197,18] := 1.0;
   DATA[197,19] := 2.0;
   DATA[197,20] := 148.808;
   DATA[197,21] := 156.0625;
   DATA[197,22] := 1.713389;
   DATA[197,23] := 959.1771;
   DATA[197,24] := 2.0;
   DATA[197,25] := 2.0;
   DATA[197,26] := 7.875737;
   DATA[197,27] := 144.7578;
   DATA[197,28] := 264.131;
   DATA[197,29] := 12.26609;
   DATA[197,30] := 1.726737;
   DATA[197,31] := 1.275778;
   DATA[197,32] := 0.7353967;
   DATA[197,33] := 0.3065048;
   DATA[197,34] := 2.0;
   DATA[197,35] := 250.8972;
   DATA[197,36] := 1.826162;
   DATA[197,37] := 189.6148;
   DATA[197,38] := 0.000128152;
   DATA[197,39] := 1.0;
   DATA[198,0] := 2.578548;
   DATA[198,1] := 527.3608;
   DATA[198,2] := 2.0;
   DATA[198,3] := 2.0;
   DATA[198,4] := 262.0802;
   DATA[198,5] := 8.391951;
   DATA[198,6] := 328.2748;
   DATA[198,7] := 2.443085;
   DATA[198,8] := 2.0;
   DATA[198,9] := 2.0;
   DATA[198,10] := 2.0;
   DATA[198,11] := 19.67796;
   DATA[198,12] := 2.213624;
   DATA[198,13] := 964.8167;
   DATA[198,14] := 1.0;
   DATA[198,15] := 2.0;
   DATA[198,16] := 1.0;
   DATA[198,17] := 1.0;
   DATA[198,18] := 1.0;
   DATA[198,19] := 2.0;
   DATA[198,20] := 148.808;
   DATA[198,21] := 156.0625;
   DATA[198,22] := 1.71262;
   DATA[198,23] := 959.3309;
   DATA[198,24] := 2.0;
   DATA[198,25] := 2.0;
   DATA[198,26] := 7.875737;
   DATA[198,27] := 144.7578;
   DATA[198,28] := 264.131;
   DATA[198,29] := 12.26609;
   DATA[198,30] := 1.726737;
   DATA[198,31] := 1.289996;
   DATA[198,32] := 0.7353967;
   DATA[198,33] := 0.3081703;
   DATA[198,34] := 2.0;
   DATA[198,35] := 250.8011;
   DATA[198,36] := 1.649953;
   DATA[198,37] := 189.5187;
   DATA[198,38] := 0.000128152;
   DATA[198,39] := 1.0;
   DATA[199,0] := 2.561573;
   DATA[199,1] := 527.1646;
   DATA[199,2] := 2.0;
   DATA[199,3] := 2.0;
   DATA[199,4] := 262.0802;
   DATA[199,5] := 8.391951;
   DATA[199,6] := 328.2748;
   DATA[199,7] := 2.442828;
   DATA[199,8] := 2.0;
   DATA[199,9] := 2.0;
   DATA[199,10] := 2.0;
   DATA[199,11] := 19.67796;
   DATA[199,12] := 2.213624;
   DATA[199,13] := 964.7767;
   DATA[199,14] := 1.0;
   DATA[199,15] := 2.0;
   DATA[199,16] := 1.0;
   DATA[199,17] := 1.0;
   DATA[199,18] := 1.0;
   DATA[199,19] := 2.0;
   DATA[199,20] := 148.808;
   DATA[199,21] := 156.0625;
   DATA[199,22] := 1.71262;
   DATA[199,23] := 959.2156;
   DATA[199,24] := 2.0;
   DATA[199,25] := 2.0;
   DATA[199,26] := 7.875737;
   DATA[199,27] := 144.7578;
   DATA[199,28] := 264.131;
   DATA[199,29] := 12.15073;
   DATA[199,30] := 1.725455;
   DATA[199,31] := 1.30114;
   DATA[199,32] := 0.7353967;
   DATA[199,33] := 0.3083624;
   DATA[199,34] := 2.0;
   DATA[199,35] := 250.785;
   DATA[199,36] := 1.649953;
   DATA[199,37] := 189.5187;
   DATA[199,38] := 0.000128152;
   DATA[199,39] := 1.0;
   DATA[200,0] := 2.54652;
   DATA[200,1] := 526.8898;
   DATA[200,2] := 2.0;
   DATA[200,3] := 2.0;
   DATA[200,4] := 262.0802;
   DATA[200,5] := 8.391951;
   DATA[200,6] := 328.2748;
   DATA[200,7] := 2.441547;
   DATA[200,8] := 2.0;
   DATA[200,9] := 2.0;
   DATA[200,10] := 2.0;
   DATA[200,11] := 19.67796;
   DATA[200,12] := 2.214906;
   DATA[200,13] := 964.9369;
   DATA[200,14] := 1.0;
   DATA[200,15] := 2.0;
   DATA[200,16] := 1.0;
   DATA[200,17] := 1.0;
   DATA[200,18] := 1.0;
   DATA[200,19] := 2.0;
   DATA[200,20] := 148.808;
   DATA[200,21] := 155.9087;
   DATA[200,22] := 1.71262;
   DATA[200,23] := 959.254;
   DATA[200,24] := 2.0;
   DATA[200,25] := 2.0;
   DATA[200,26] := 7.875737;
   DATA[200,27] := 144.7578;
   DATA[200,28] := 264.131;
   DATA[200,29] := 12.03538;
   DATA[200,30] := 1.72507;
   DATA[200,31] := 1.30178;
   DATA[200,32] := 0.7353967;
   DATA[200,33] := 0.3083624;
   DATA[200,34] := 2.0;
   DATA[200,35] := 250.785;
   DATA[200,36] := 1.649953;
   DATA[200,37] := 189.5187;
   DATA[200,38] := 0.000128152;
   DATA[200,39] := 1.0;
   DATA[201,0] := 2.52282;
   DATA[201,1] := 526.772;
   DATA[201,2] := 2.0;
   DATA[201,3] := 2.0;
   DATA[201,4] := 262.0802;
   DATA[201,5] := 8.391951;
   DATA[201,6] := 328.2748;
   DATA[201,7] := 2.440137;
   DATA[201,8] := 2.0;
   DATA[201,9] := 2.0;
   DATA[201,10] := 2.0;
   DATA[201,11] := 19.67796;
   DATA[201,12] := 2.214906;
   DATA[201,13] := 965.0571;
   DATA[201,14] := 1.0;
   DATA[201,15] := 2.0;
   DATA[201,16] := 1.0;
   DATA[201,17] := 1.0;
   DATA[201,18] := 1.0;
   DATA[201,19] := 2.0;
   DATA[201,20] := 148.808;
   DATA[201,21] := 155.9087;
   DATA[201,22] := 1.71262;
   DATA[201,23] := 959.3309;
   DATA[201,24] := 2.0;
   DATA[201,25] := 2.0;
   DATA[201,26] := 7.875737;
   DATA[201,27] := 144.7578;
   DATA[201,28] := 264.131;
   DATA[201,29] := 12.03538;
   DATA[201,30] := 1.724814;
   DATA[201,31] := 1.311259;
   DATA[201,32] := 0.7353967;
   DATA[201,33] := 0.3083624;
   DATA[201,34] := 2.0;
   DATA[201,35] := 250.785;
   DATA[201,36] := 1.778105;
   DATA[201,37] := 189.5187;
   DATA[201,38] := 0.000128152;
   DATA[201,39] := 1.0;
   DATA[202,0] := 2.503283;
   DATA[202,1] := 526.4973;
   DATA[202,2] := 2.0;
   DATA[202,3] := 2.0;
   DATA[202,4] := 262.0802;
   DATA[202,5] := 8.394835;
   DATA[202,6] := 328.2748;
   DATA[202,7] := 2.440137;
   DATA[202,8] := 2.0;
   DATA[202,9] := 2.0;
   DATA[202,10] := 2.0;
   DATA[202,11] := 19.67796;
   DATA[202,12] := 2.212343;
   DATA[202,13] := 965.0571;
   DATA[202,14] := 1.0;
   DATA[202,15] := 2.0;
   DATA[202,16] := 1.0;
   DATA[202,17] := 1.0;
   DATA[202,18] := 1.0;
   DATA[202,19] := 2.0;
   DATA[202,20] := 148.808;
   DATA[202,21] := 155.9087;
   DATA[202,22] := 1.714798;
   DATA[202,23] := 959.2156;
   DATA[202,24] := 2.0;
   DATA[202,25] := 2.0;
   DATA[202,26] := 7.875737;
   DATA[202,27] := 144.7578;
   DATA[202,28] := 264.131;
   DATA[202,29] := 12.03538;
   DATA[202,30] := 1.724814;
   DATA[202,31] := 1.305623;
   DATA[202,32] := 0.7353967;
   DATA[202,33] := 0.3083624;
   DATA[202,34] := 2.0;
   DATA[202,35] := 250.785;
   DATA[202,36] := 1.778105;
   DATA[202,37] := 189.5187;
   DATA[202,38] := 0.000128152;
   DATA[202,39] := 1.0;
   DATA[203,0] := 2.485027;
   DATA[203,1] := 526.301;
   DATA[203,2] := 2.0;
   DATA[203,3] := 2.0;
   DATA[203,4] := 262.0802;
   DATA[203,5] := 8.394835;
   DATA[203,6] := 328.2748;
   DATA[203,7] := 2.440137;
   DATA[203,8] := 2.0;
   DATA[203,9] := 2.0;
   DATA[203,10] := 2.0;
   DATA[203,11] := 19.70037;
   DATA[203,12] := 2.212343;
   DATA[203,13] := 965.3775;
   DATA[203,14] := 1.0;
   DATA[203,15] := 2.0;
   DATA[203,16] := 1.0;
   DATA[203,17] := 1.0;
   DATA[203,18] := 1.0;
   DATA[203,19] := 2.0;
   DATA[203,20] := 148.808;
   DATA[203,21] := 155.9087;
   DATA[203,22] := 1.717233;
   DATA[203,23] := 959.2156;
   DATA[203,24] := 2.0;
   DATA[203,25] := 2.0;
   DATA[203,26] := 7.875737;
   DATA[203,27] := 144.7578;
   DATA[203,28] := 264.131;
   DATA[203,29] := 12.03538;
   DATA[203,30] := 1.726096;
   DATA[203,31] := 1.292558;
   DATA[203,32] := 0.7353967;
   DATA[203,33] := 0.3083624;
   DATA[203,34] := 2.0;
   DATA[203,35] := 250.785;
   DATA[203,36] := 1.778105;
   DATA[203,37] := 189.5187;
   DATA[203,38] := 0.000128152;
   DATA[203,39] := 1.0;
   DATA[204,0] := 2.467092;
   DATA[204,1] := 526.0262;
   DATA[204,2] := 2.0;
   DATA[204,3] := 2.0;
   DATA[204,4] := 262.0802;
   DATA[204,5] := 8.394835;
   DATA[204,6] := 328.2748;
   DATA[204,7] := 2.441547;
   DATA[204,8] := 2.0;
   DATA[204,9] := 2.0;
   DATA[204,10] := 2.0;
   DATA[204,11] := 19.73238;
   DATA[204,12] := 2.209525;
   DATA[204,13] := 965.4576;
   DATA[204,14] := 1.0;
   DATA[204,15] := 2.0;
   DATA[204,16] := 1.0;
   DATA[204,17] := 1.0;
   DATA[204,18] := 1.0;
   DATA[204,19] := 2.0;
   DATA[204,20] := 148.808;
   DATA[204,21] := 155.9087;
   DATA[204,22] := 1.717489;
   DATA[204,23] := 958.8695;
   DATA[204,24] := 2.0;
   DATA[204,25] := 2.0;
   DATA[204,26] := 7.875737;
   DATA[204,27] := 144.7578;
   DATA[204,28] := 264.131;
   DATA[204,29] := 12.03538;
   DATA[204,30] := 1.726096;
   DATA[204,31] := 1.292174;
   DATA[204,32] := 0.7353967;
   DATA[204,33] := 0.3083624;
   DATA[204,34] := 2.0;
   DATA[204,35] := 250.8812;
   DATA[204,36] := 1.778105;
   DATA[204,37] := 189.5187;
   DATA[204,38] := 0.000128152;
   DATA[204,39] := 1.0;
   DATA[205,0] := 2.452679;
   DATA[205,1] := 526.0262;
   DATA[205,2] := 2.0;
   DATA[205,3] := 2.0;
   DATA[205,4] := 262.0802;
   DATA[205,5] := 8.394835;
   DATA[205,6] := 328.2748;
   DATA[205,7] := 2.441547;
   DATA[205,8] := 2.0;
   DATA[205,9] := 2.0;
   DATA[205,10] := 2.0;
   DATA[205,11] := 19.73238;
   DATA[205,12] := 2.209269;
   DATA[205,13] := 965.5778;
   DATA[205,14] := 1.0;
   DATA[205,15] := 2.0;
   DATA[205,16] := 1.0;
   DATA[205,17] := 1.0;
   DATA[205,18] := 1.0;
   DATA[205,19] := 2.0;
   DATA[205,20] := 148.808;
   DATA[205,21] := 155.9087;
   DATA[205,22] := 1.717489;
   DATA[205,23] := 958.8311;
   DATA[205,24] := 2.0;
   DATA[205,25] := 2.0;
   DATA[205,26] := 7.875737;
   DATA[205,27] := 144.7578;
   DATA[205,28] := 264.131;
   DATA[205,29] := 12.03538;
   DATA[205,30] := 1.726737;
   DATA[205,31] := 1.282311;
   DATA[205,32] := 0.7353967;
   DATA[205,33] := 0.3083624;
   DATA[205,34] := 2.0;
   DATA[205,35] := 250.9132;
   DATA[205,36] := 1.69801;
   DATA[205,37] := 189.6629;
   DATA[205,38] := 0.000128152;
   DATA[205,39] := 1.0;
   DATA[206,0] := 2.436345;
   DATA[206,1] := 525.83;
   DATA[206,2] := 2.0;
   DATA[206,3] := 2.0;
   DATA[206,4] := 262.0802;
   DATA[206,5] := 8.394835;
   DATA[206,6] := 328.2748;
   DATA[206,7] := 2.4427;
   DATA[206,8] := 2.0;
   DATA[206,9] := 2.0;
   DATA[206,10] := 2.0;
   DATA[206,11] := 19.67476;
   DATA[206,12] := 2.208372;
   DATA[206,13] := 965.6178;
   DATA[206,14] := 1.0;
   DATA[206,15] := 2.0;
   DATA[206,16] := 1.0;
   DATA[206,17] := 1.0;
   DATA[206,18] := 1.0;
   DATA[206,19] := 2.0;
   DATA[206,20] := 148.808;
   DATA[206,21] := 155.9087;
   DATA[206,22] := 1.717489;
   DATA[206,23] := 958.6388;
   DATA[206,24] := 2.0;
   DATA[206,25] := 2.0;
   DATA[206,26] := 7.875737;
   DATA[206,27] := 144.7578;
   DATA[206,28] := 264.131;
   DATA[206,29] := 12.03538;
   DATA[206,30] := 1.726737;
   DATA[206,31] := 1.281798;
   DATA[206,32] := 0.7353967;
   DATA[206,33] := 0.3083624;
   DATA[206,34] := 2.0;
   DATA[206,35] := 250.9132;
   DATA[206,36] := 1.69801;
   DATA[206,37] := 189.759;
   DATA[206,38] := 0.000128152;
   DATA[206,39] := 1.0;
   DATA[207,0] := 2.428979;
   DATA[207,1] := 525.4767;
   DATA[207,2] := 2.0;
   DATA[207,3] := 2.0;
   DATA[207,4] := 262.0802;
   DATA[207,5] := 8.394835;
   DATA[207,6] := 328.2748;
   DATA[207,7] := 2.443469;
   DATA[207,8] := 2.0;
   DATA[207,9] := 2.0;
   DATA[207,10] := 2.0;
   DATA[207,11] := 19.64594;
   DATA[207,12] := 2.207731;
   DATA[207,13] := 966.1385;
   DATA[207,14] := 1.0;
   DATA[207,15] := 2.0;
   DATA[207,16] := 1.0;
   DATA[207,17] := 1.0;
   DATA[207,18] := 1.0;
   DATA[207,19] := 2.0;
   DATA[207,20] := 148.808;
   DATA[207,21] := 155.9087;
   DATA[207,22] := 1.716464;
   DATA[207,23] := 958.6388;
   DATA[207,24] := 2.0;
   DATA[207,25] := 2.0;
   DATA[207,26] := 7.875737;
   DATA[207,27] := 144.7578;
   DATA[207,28] := 264.131;
   DATA[207,29] := 12.03538;
   DATA[207,30] := 1.726737;
   DATA[207,31] := 1.281542;
   DATA[207,32] := 0.7353967;
   DATA[207,33] := 0.3083624;
   DATA[207,34] := 2.0;
   DATA[207,35] := 250.9132;
   DATA[207,36] := 1.69801;
   DATA[207,37] := 189.759;
   DATA[207,38] := 0.000128152;
   DATA[207,39] := 1.0;
   DATA[208,0] := 2.423534;
   DATA[208,1] := 525.5944;
   DATA[208,2] := 2.0;
   DATA[208,3] := 2.0;
   DATA[208,4] := 262.0802;
   DATA[208,5] := 8.394835;
   DATA[208,6] := 328.2748;
   DATA[208,7] := 2.443725;
   DATA[208,8] := 2.0;
   DATA[208,9] := 2.0;
   DATA[208,10] := 2.0;
   DATA[208,11] := 19.64594;
   DATA[208,12] := 2.207731;
   DATA[208,13] := 966.3788;
   DATA[208,14] := 1.0;
   DATA[208,15] := 2.0;
   DATA[208,16] := 1.0;
   DATA[208,17] := 1.0;
   DATA[208,18] := 1.0;
   DATA[208,19] := 2.0;
   DATA[208,20] := 148.808;
   DATA[208,21] := 155.9087;
   DATA[208,22] := 1.716464;
   DATA[208,23] := 958.1774;
   DATA[208,24] := 2.0;
   DATA[208,25] := 2.0;
   DATA[208,26] := 7.875737;
   DATA[208,27] := 144.7578;
   DATA[208,28] := 264.131;
   DATA[208,29] := 12.03538;
   DATA[208,30] := 1.726737;
   DATA[208,31] := 1.281542;
   DATA[208,32] := 0.7353967;
   DATA[208,33] := 0.3083624;
   DATA[208,34] := 2.0;
   DATA[208,35] := 250.9132;
   DATA[208,36] := 1.69801;
   DATA[208,37] := 189.759;
   DATA[208,38] := 0.000128152;
   DATA[208,39] := 1.0;
   DATA[209,0] := 2.423534;
   DATA[209,1] := 525.6729;
   DATA[209,2] := 2.0;
   DATA[209,3] := 2.0;
   DATA[209,4] := 262.0802;
   DATA[209,5] := 8.394835;
   DATA[209,6] := 328.2748;
   DATA[209,7] := 2.443725;
   DATA[209,8] := 2.0;
   DATA[209,9] := 2.0;
   DATA[209,10] := 2.0;
   DATA[209,11] := 19.67476;
   DATA[209,12] := 2.207731;
   DATA[209,13] := 966.4189;
   DATA[209,14] := 1.0;
   DATA[209,15] := 2.0;
   DATA[209,16] := 1.0;
   DATA[209,17] := 1.0;
   DATA[209,18] := 1.0;
   DATA[209,19] := 2.0;
   DATA[209,20] := 148.808;
   DATA[209,21] := 155.9087;
   DATA[209,22] := 1.716464;
   DATA[209,23] := 958.1774;
   DATA[209,24] := 2.0;
   DATA[209,25] := 2.0;
   DATA[209,26] := 7.876058;
   DATA[209,27] := 144.7578;
   DATA[209,28] := 264.131;
   DATA[209,29] := 12.03538;
   DATA[209,30] := 1.726737;
   DATA[209,31] := 1.271551;
   DATA[209,32] := 0.7353967;
   DATA[209,33] := 0.3083624;
   DATA[209,34] := 2.0;
   DATA[209,35] := 250.9132;
   DATA[209,36] := 1.69801;
   DATA[209,37] := 189.759;
   DATA[209,38] := 0.000128152;
   DATA[209,39] := 1.0;
   DATA[210,0] := 2.45428;
   DATA[210,1] := 525.7907;
   DATA[210,2] := 2.0;
   DATA[210,3] := 2.0;
   DATA[210,4] := 262.0802;
   DATA[210,5] := 8.394835;
   DATA[210,6] := 328.2748;
   DATA[210,7] := 2.442828;
   DATA[210,8] := 2.0;
   DATA[210,9] := 2.0;
   DATA[210,10] := 2.0;
   DATA[210,11] := 19.69396;
   DATA[210,12] := 2.209653;
   DATA[210,13] := 966.8595;
   DATA[210,14] := 1.0;
   DATA[210,15] := 2.0;
   DATA[210,16] := 1.0;
   DATA[210,17] := 1.0;
   DATA[210,18] := 1.0;
   DATA[210,19] := 2.0;
   DATA[210,20] := 148.808;
   DATA[210,21] := 155.9087;
   DATA[210,22] := 1.716464;
   DATA[210,23] := 958.1389;
   DATA[210,24] := 2.0;
   DATA[210,25] := 2.0;
   DATA[210,26] := 7.876058;
   DATA[210,27] := 144.7578;
   DATA[210,28] := 264.131;
   DATA[210,29] := 12.03538;
   DATA[210,30] := 1.726737;
   DATA[210,31] := 1.261688;
   DATA[210,32] := 0.7353967;
   DATA[210,33] := 0.3083624;
   DATA[210,34] := 2.0;
   DATA[210,35] := 251.0254;
   DATA[210,36] := 1.69801;
   DATA[210,37] := 189.759;
   DATA[210,38] := 0.000128152;
   DATA[210,39] := 1.0;
   DATA[211,0] := 2.45428;
   DATA[211,1] := 525.7907;
   DATA[211,2] := 2.0;
   DATA[211,3] := 2.0;
   DATA[211,4] := 262.0802;
   DATA[211,5] := 8.394835;
   DATA[211,6] := 328.2748;
   DATA[211,7] := 2.442828;
   DATA[211,8] := 2.0;
   DATA[211,9] := 2.0;
   DATA[211,10] := 2.0;
   DATA[211,11] := 19.69396;
   DATA[211,12] := 2.209653;
   DATA[211,13] := 966.8595;
   DATA[211,14] := 1.0;
   DATA[211,15] := 2.0;
   DATA[211,16] := 1.0;
   DATA[211,17] := 1.0;
   DATA[211,18] := 1.0;
   DATA[211,19] := 2.0;
   DATA[211,20] := 148.808;
   DATA[211,21] := 155.9087;
   DATA[211,22] := 1.716464;
   DATA[211,23] := 958.1389;
   DATA[211,24] := 2.0;
   DATA[211,25] := 2.0;
   DATA[211,26] := 7.876058;
   DATA[211,27] := 144.7578;
   DATA[211,28] := 264.131;
   DATA[211,29] := 12.03538;
   DATA[211,30] := 1.726737;
   DATA[211,31] := 1.261688;
   DATA[211,32] := 0.7353967;
   DATA[211,33] := 0.3083624;
   DATA[211,34] := 2.0;
   DATA[211,35] := 251.0254;
   DATA[211,36] := 1.69801;
   DATA[211,37] := 189.759;
   DATA[211,38] := 0.000128152;
   DATA[211,39] := 1.0;
   DATA[212,0] := 2.490792;
   DATA[212,1] := 525.6729;
   DATA[212,2] := 2.0;
   DATA[212,3] := 2.0;
   DATA[212,4] := 262.0802;
   DATA[212,5] := 8.394835;
   DATA[212,6] := 328.2748;
   DATA[212,7] := 2.440521;
   DATA[212,8] := 2.0;
   DATA[212,9] := 2.0;
   DATA[212,10] := 2.0;
   DATA[212,11] := 19.73878;
   DATA[212,12] := 2.209653;
   DATA[212,13] := 966.9396;
   DATA[212,14] := 1.0;
   DATA[212,15] := 2.0;
   DATA[212,16] := 1.0;
   DATA[212,17] := 1.0;
   DATA[212,18] := 1.0;
   DATA[212,19] := 2.0;
   DATA[212,20] := 148.808;
   DATA[212,21] := 155.9087;
   DATA[212,22] := 1.716464;
   DATA[212,23] := 958.2158;
   DATA[212,24] := 2.0;
   DATA[212,25] := 2.0;
   DATA[212,26] := 7.876058;
   DATA[212,27] := 144.7578;
   DATA[212,28] := 264.131;
   DATA[212,29] := 12.26609;
   DATA[212,30] := 1.726737;
   DATA[212,31] := 1.26758;
   DATA[212,32] := 0.7353967;
   DATA[212,33] := 0.3083624;
   DATA[212,34] := 2.0;
   DATA[212,35] := 251.1055;
   DATA[212,36] := 1.69801;
   DATA[212,37] := 189.759;
   DATA[212,38] := 0.000128152;
   DATA[212,39] := 1.0;
   DATA[213,0] := 2.535951;
   DATA[213,1] := 526.1047;
   DATA[213,2] := 2.0;
   DATA[213,3] := 2.0;
   DATA[213,4] := 262.0802;
   DATA[213,5] := 8.394835;
   DATA[213,6] := 328.2748;
   DATA[213,7] := 2.440521;
   DATA[213,8] := 2.0;
   DATA[213,9] := 2.0;
   DATA[213,10] := 2.0;
   DATA[213,11] := 19.74838;
   DATA[213,12] := 2.209653;
   DATA[213,13] := 967.0598;
   DATA[213,14] := 1.0;
   DATA[213,15] := 2.0;
   DATA[213,16] := 1.0;
   DATA[213,17] := 1.0;
   DATA[213,18] := 1.0;
   DATA[213,19] := 2.0;
   DATA[213,20] := 148.808;
   DATA[213,21] := 155.7806;
   DATA[213,22] := 1.715311;
   DATA[213,23] := 957.8698;
   DATA[213,24] := 2.0;
   DATA[213,25] := 2.0;
   DATA[213,26] := 7.876058;
   DATA[213,27] := 144.7578;
   DATA[213,28] := 264.131;
   DATA[213,29] := 12.26609;
   DATA[213,30] := 1.726737;
   DATA[213,31] := 1.272576;
   DATA[213,32] := 0.7353967;
   DATA[213,33] := 0.3083624;
   DATA[213,34] := 2.0;
   DATA[213,35] := 251.1055;
   DATA[213,36] := 1.69801;
   DATA[213,37] := 189.759;
   DATA[213,38] := 0.000128152;
   DATA[213,39] := 1.0;
   DATA[214,0] := 2.5699;
   DATA[214,1] := 526.2617;
   DATA[214,2] := 2.0;
   DATA[214,3] := 2.0;
   DATA[214,4] := 262.0802;
   DATA[214,5] := 8.394835;
   DATA[214,6] := 328.2748;
   DATA[214,7] := 2.440521;
   DATA[214,8] := 2.0;
   DATA[214,9] := 2.0;
   DATA[214,10] := 2.0;
   DATA[214,11] := 19.74838;
   DATA[214,12] := 2.209653;
   DATA[214,13] := 967.0197;
   DATA[214,14] := 1.0;
   DATA[214,15] := 2.0;
   DATA[214,16] := 1.0;
   DATA[214,17] := 1.0;
   DATA[214,18] := 1.0;
   DATA[214,19] := 2.0;
   DATA[214,20] := 148.808;
   DATA[214,21] := 155.7806;
   DATA[214,22] := 1.715183;
   DATA[214,23] := 957.4853;
   DATA[214,24] := 2.0;
   DATA[214,25] := 2.0;
   DATA[214,26] := 7.876058;
   DATA[214,27] := 144.7578;
   DATA[214,28] := 264.131;
   DATA[214,29] := 12.26609;
   DATA[214,30] := 1.726737;
   DATA[214,31] := 1.282439;
   DATA[214,32] := 0.7353967;
   DATA[214,33] := 0.3083624;
   DATA[214,34] := 2.0;
   DATA[214,35] := 251.1055;
   DATA[214,36] := 1.746067;
   DATA[214,37] := 189.759;
   DATA[214,38] := 0.000128152;
   DATA[214,39] := 1.0;
   DATA[215,0] := 2.611536;
   DATA[215,1] := 526.8113;
   DATA[215,2] := 2.0;
   DATA[215,3] := 2.0;
   DATA[215,4] := 262.0802;
   DATA[215,5] := 8.394835;
   DATA[215,6] := 328.2748;
   DATA[215,7] := 2.440521;
   DATA[215,8] := 2.0;
   DATA[215,9] := 2.0;
   DATA[215,10] := 2.0;
   DATA[215,11] := 19.74838;
   DATA[215,12] := 2.210934;
   DATA[215,13] := 967.22;
   DATA[215,14] := 1.0;
   DATA[215,15] := 2.0;
   DATA[215,16] := 1.0;
   DATA[215,17] := 1.0;
   DATA[215,18] := 1.0;
   DATA[215,19] := 2.0;
   DATA[215,20] := 148.808;
   DATA[215,21] := 155.7806;
   DATA[215,22] := 1.715183;
   DATA[215,23] := 957.4853;
   DATA[215,24] := 2.0;
   DATA[215,25] := 2.0;
   DATA[215,26] := 7.876058;
   DATA[215,27] := 144.7578;
   DATA[215,28] := 264.131;
   DATA[215,29] := 12.26609;
   DATA[215,30] := 1.726737;
   DATA[215,31] := 1.291533;
   DATA[215,32] := 0.7353967;
   DATA[215,33] := 0.3083624;
   DATA[215,34] := 2.0;
   DATA[215,35] := 251.1055;
   DATA[215,36] := 1.746067;
   DATA[215,37] := 189.759;
   DATA[215,38] := 0.000128152;
   DATA[215,39] := 1.0;
   DATA[216,0] := 2.633315;
   DATA[216,1] := 527.3608;
   DATA[216,2] := 2.0;
   DATA[216,3] := 2.0;
   DATA[216,4] := 262.0802;
   DATA[216,5] := 8.392912;
   DATA[216,6] := 328.2748;
   DATA[216,7] := 2.440521;
   DATA[216,8] := 2.0;
   DATA[216,9] := 2.0;
   DATA[216,10] := 2.0;
   DATA[216,11] := 19.72598;
   DATA[216,12] := 2.212343;
   DATA[216,13] := 967.0197;
   DATA[216,14] := 1.0;
   DATA[216,15] := 2.0;
   DATA[216,16] := 1.0;
   DATA[216,17] := 1.0;
   DATA[216,18] := 1.0;
   DATA[216,19] := 2.0;
   DATA[216,20] := 148.808;
   DATA[216,21] := 155.7806;
   DATA[216,22] := 1.717746;
   DATA[216,23] := 957.7544;
   DATA[216,24] := 2.0;
   DATA[216,25] := 2.0;
   DATA[216,26] := 7.876058;
   DATA[216,27] := 144.7578;
   DATA[216,28] := 264.131;
   DATA[216,29] := 12.26609;
   DATA[216,30] := 1.72725;
   DATA[216,31] := 1.286922;
   DATA[216,32] := 0.7353967;
   DATA[216,33] := 0.3074016;
   DATA[216,34] := 2.0;
   DATA[216,35] := 251.1055;
   DATA[216,36] := 1.746067;
   DATA[216,37] := 189.759;
   DATA[216,38] := 0.000128152;
   DATA[216,39] := 1.0;
   DATA[217,0] := 2.652211;
   DATA[217,1] := 528.1459;
   DATA[217,2] := 2.0;
   DATA[217,3] := 2.0;
   DATA[217,4] := 262.0802;
   DATA[217,5] := 8.391951;
   DATA[217,6] := 328.2748;
   DATA[217,7] := 2.440265;
   DATA[217,8] := 2.0;
   DATA[217,9] := 2.0;
   DATA[217,10] := 2.0;
   DATA[217,11] := 19.71957;
   DATA[217,12] := 2.21324;
   DATA[217,13] := 967.3802;
   DATA[217,14] := 1.0;
   DATA[217,15] := 2.0;
   DATA[217,16] := 1.0;
   DATA[217,17] := 1.0;
   DATA[217,18] := 1.0;
   DATA[217,19] := 2.0;
   DATA[217,20] := 148.808;
   DATA[217,21] := 155.7806;
   DATA[217,22] := 1.717746;
   DATA[217,23] := 957.4468;
   DATA[217,24] := 2.0;
   DATA[217,25] := 2.0;
   DATA[217,26] := 7.876058;
   DATA[217,27] := 144.7578;
   DATA[217,28] := 264.131;
   DATA[217,29] := 12.26609;
   DATA[217,30] := 1.72725;
   DATA[217,31] := 1.286922;
   DATA[217,32] := 0.7353967;
   DATA[217,33] := 0.3066329;
   DATA[217,34] := 2.0;
   DATA[217,35] := 251.1055;
   DATA[217,36] := 1.746067;
   DATA[217,37] := 189.8231;
   DATA[217,38] := 0.000128152;
   DATA[217,39] := 1.0;
   DATA[218,0] := 2.655414;
   DATA[218,1] := 528.2636;
   DATA[218,2] := 2.0;
   DATA[218,3] := 2.0;
   DATA[218,4] := 262.0802;
   DATA[218,5] := 8.391951;
   DATA[218,6] := 328.2748;
   DATA[218,7] := 2.440265;
   DATA[218,8] := 2.0;
   DATA[218,9] := 2.0;
   DATA[218,10] := 2.0;
   DATA[218,11] := 19.71957;
   DATA[218,12] := 2.214649;
   DATA[218,13] := 967.26;
   DATA[218,14] := 1.0;
   DATA[218,15] := 2.0;
   DATA[218,16] := 1.0;
   DATA[218,17] := 1.0;
   DATA[218,18] := 1.0;
   DATA[218,19] := 2.0;
   DATA[218,20] := 148.808;
   DATA[218,21] := 155.7806;
   DATA[218,22] := 1.719027;
   DATA[218,23] := 957.4468;
   DATA[218,24] := 2.0;
   DATA[218,25] := 2.0;
   DATA[218,26] := 7.876058;
   DATA[218,27] := 144.8347;
   DATA[218,28] := 264.131;
   DATA[218,29] := 12.07383;
   DATA[218,30] := 1.728147;
   DATA[218,31] := 1.284104;
   DATA[218,32] := 0.7353967;
   DATA[218,33] := 0.3066329;
   DATA[218,34] := 2.0;
   DATA[218,35] := 251.1856;
   DATA[218,36] := 1.746067;
   DATA[218,37] := 189.9193;
   DATA[218,38] := 0.000128152;
   DATA[218,39] := 1.0;
   DATA[219,0] := 2.642603;
   DATA[219,1] := 528.4207;
   DATA[219,2] := 2.0;
   DATA[219,3] := 2.0;
   DATA[219,4] := 262.0802;
   DATA[219,5] := 8.391951;
   DATA[219,6] := 328.2748;
   DATA[219,7] := 2.440265;
   DATA[219,8] := 2.0;
   DATA[219,9] := 2.0;
   DATA[219,10] := 2.0;
   DATA[219,11] := 19.71957;
   DATA[219,12] := 2.210678;
   DATA[219,13] := 967.0197;
   DATA[219,14] := 1.0;
   DATA[219,15] := 2.0;
   DATA[219,16] := 1.0;
   DATA[219,17] := 1.0;
   DATA[219,18] := 1.0;
   DATA[219,19] := 2.0;
   DATA[219,20] := 148.808;
   DATA[219,21] := 155.7806;
   DATA[219,22] := 1.719156;
   DATA[219,23] := 957.9467;
   DATA[219,24] := 2.0;
   DATA[219,25] := 2.0;
   DATA[219,26] := 7.876058;
   DATA[219,27] := 144.8347;
   DATA[219,28] := 264.131;
   DATA[219,29] := 12.07383;
   DATA[219,30] := 1.728531;
   DATA[219,31] := 1.282567;
   DATA[219,32] := 0.7353967;
   DATA[219,33] := 0.3066329;
   DATA[219,34] := 2.0;
   DATA[219,35] := 251.2977;
   DATA[219,36] := 1.746067;
   DATA[219,37] := 190.0634;
   DATA[219,38] := 0.000128152;
   DATA[219,39] := 1.0;
   DATA[220,0] := 2.626589;
   DATA[220,1] := 528.4207;
   DATA[220,2] := 2.0;
   DATA[220,3] := 2.0;
   DATA[220,4] := 262.0802;
   DATA[220,5] := 8.391951;
   DATA[220,6] := 328.2748;
   DATA[220,7] := 2.440265;
   DATA[220,8] := 2.0;
   DATA[220,9] := 2.0;
   DATA[220,10] := 2.0;
   DATA[220,11] := 19.71957;
   DATA[220,12] := 2.209397;
   DATA[220,13] := 967.22;
   DATA[220,14] := 1.0;
   DATA[220,15] := 2.0;
   DATA[220,16] := 1.0;
   DATA[220,17] := 1.0;
   DATA[220,18] := 1.0;
   DATA[220,19] := 2.0;
   DATA[220,20] := 148.808;
   DATA[220,21] := 155.7806;
   DATA[220,22] := 1.719156;
   DATA[220,23] := 958.3696;
   DATA[220,24] := 2.0;
   DATA[220,25] := 2.0;
   DATA[220,26] := 7.876058;
   DATA[220,27] := 144.8347;
   DATA[220,28] := 264.131;
   DATA[220,29] := 12.07383;
   DATA[220,30] := 1.731095;
   DATA[220,31] := 1.289868;
   DATA[220,32] := 0.7353967;
   DATA[220,33] := 0.3066329;
   DATA[220,34] := 2.0;
   DATA[220,35] := 251.2977;
   DATA[220,36] := 1.746067;
   DATA[220,37] := 190.0634;
   DATA[220,38] := 0.000128152;
   DATA[220,39] := 1.0;
   DATA[221,0] := 2.619223;
   DATA[221,1] := 528.1459;
   DATA[221,2] := 2.0;
   DATA[221,3] := 2.0;
   DATA[221,4] := 262.0802;
   DATA[221,5] := 8.391951;
   DATA[221,6] := 328.2748;
   DATA[221,7] := 2.440265;
   DATA[221,8] := 2.0;
   DATA[221,9] := 2.0;
   DATA[221,10] := 2.0;
   DATA[221,11] := 19.71957;
   DATA[221,12] := 2.209397;
   DATA[221,13] := 967.1398;
   DATA[221,14] := 1.0;
   DATA[221,15] := 2.0;
   DATA[221,16] := 1.0;
   DATA[221,17] := 1.0;
   DATA[221,18] := 1.0;
   DATA[221,19] := 2.0;
   DATA[221,20] := 148.808;
   DATA[221,21] := 155.7806;
   DATA[221,22] := 1.719156;
   DATA[221,23] := 958.5619;
   DATA[221,24] := 2.0;
   DATA[221,25] := 2.0;
   DATA[221,26] := 7.876058;
   DATA[221,27] := 144.8347;
   DATA[221,28] := 264.131;
   DATA[221,29] := 12.07383;
   DATA[221,30] := 1.731095;
   DATA[221,31] := 1.292046;
   DATA[221,32] := 0.7353967;
   DATA[221,33] := 0.3066329;
   DATA[221,34] := 2.0;
   DATA[221,35] := 251.2977;
   DATA[221,36] := 1.746067;
   DATA[221,37] := 190.0634;
   DATA[221,38] := 0.000128152;
   DATA[221,39] := 1.0;
   DATA[222,0] := 2.616981;
   DATA[222,1] := 527.8318;
   DATA[222,2] := 2.0;
   DATA[222,3] := 2.0;
   DATA[222,4] := 262.0802;
   DATA[222,5] := 8.391951;
   DATA[222,6] := 328.2748;
   DATA[222,7] := 2.440265;
   DATA[222,8] := 2.0;
   DATA[222,9] := 2.0;
   DATA[222,10] := 2.0;
   DATA[222,11] := 19.68756;
   DATA[222,12] := 2.211575;
   DATA[222,13] := 967.3802;
   DATA[222,14] := 1.0;
   DATA[222,15] := 2.0;
   DATA[222,16] := 1.0;
   DATA[222,17] := 1.0;
   DATA[222,18] := 1.0;
   DATA[222,19] := 2.0;
   DATA[222,20] := 148.808;
   DATA[222,21] := 155.7806;
   DATA[222,22] := 1.719156;
   DATA[222,23] := 958.7157;
   DATA[222,24] := 2.0;
   DATA[222,25] := 2.0;
   DATA[222,26] := 7.876058;
   DATA[222,27] := 144.8347;
   DATA[222,28] := 264.131;
   DATA[222,29] := 12.07383;
   DATA[222,30] := 1.731095;
   DATA[222,31] := 1.304342;
   DATA[222,32] := 0.7353967;
   DATA[222,33] := 0.3074016;
   DATA[222,34] := 2.0;
   DATA[222,35] := 251.2977;
   DATA[222,36] := 1.746067;
   DATA[222,37] := 190.0634;
   DATA[222,38] := 0.000128152;
   DATA[222,39] := 1.0;
   DATA[223,0] := 2.598725;
   DATA[223,1] := 527.243;
   DATA[223,2] := 2.0;
   DATA[223,3] := 2.0;
   DATA[223,4] := 262.0802;
   DATA[223,5] := 8.391951;
   DATA[223,6] := 328.2748;
   DATA[223,7] := 2.440265;
   DATA[223,8] := 2.0;
   DATA[223,9] := 2.0;
   DATA[223,10] := 2.0;
   DATA[223,11] := 19.68756;
   DATA[223,12] := 2.212728;
   DATA[223,13] := 967.3802;
   DATA[223,14] := 1.0;
   DATA[223,15] := 2.0;
   DATA[223,16] := 1.0;
   DATA[223,17] := 1.0;
   DATA[223,18] := 1.0;
   DATA[223,19] := 2.0;
   DATA[223,20] := 148.808;
   DATA[223,21] := 155.7806;
   DATA[223,22] := 1.720053;
   DATA[223,23] := 958.9849;
   DATA[223,24] := 2.0;
   DATA[223,25] := 2.0;
   DATA[223,26] := 7.876058;
   DATA[223,27] := 144.8347;
   DATA[223,28] := 264.131;
   DATA[223,29] := 12.07383;
   DATA[223,30] := 1.731095;
   DATA[223,31] := 1.311131;
   DATA[223,32] := 0.7353967;
   DATA[223,33] := 0.3084905;
   DATA[223,34] := 2.0;
   DATA[223,35] := 251.522;
   DATA[223,36] := 1.746067;
   DATA[223,37] := 190.0634;
   DATA[223,38] := 0.000128152;
   DATA[223,39] := 1.0;
   DATA[224,0] := 2.584313;
   DATA[224,1] := 526.6542;
   DATA[224,2] := 2.0;
   DATA[224,3] := 2.0;
   DATA[224,4] := 262.0802;
   DATA[224,5] := 8.391951;
   DATA[224,6] := 328.2748;
   DATA[224,7] := 2.440265;
   DATA[224,8] := 2.0;
   DATA[224,9] := 2.0;
   DATA[224,10] := 2.0;
   DATA[224,11] := 19.73558;
   DATA[224,12] := 2.212728;
   DATA[224,13] := 967.0598;
   DATA[224,14] := 1.0;
   DATA[224,15] := 2.0;
   DATA[224,16] := 1.0;
   DATA[224,17] := 1.0;
   DATA[224,18] := 1.0;
   DATA[224,19] := 2.0;
   DATA[224,20] := 148.808;
   DATA[224,21] := 155.7806;
   DATA[224,22] := 1.720565;
   DATA[224,23] := 959.254;
   DATA[224,24] := 2.0;
   DATA[224,25] := 2.0;
   DATA[224,26] := 7.876058;
   DATA[224,27] := 144.8347;
   DATA[224,28] := 264.131;
   DATA[224,29] := 12.07383;
   DATA[224,30] := 1.731095;
   DATA[224,31] := 1.312284;
   DATA[224,32] := 0.7353967;
   DATA[224,33] := 0.3084905;
   DATA[224,34] := 2.0;
   DATA[224,35] := 251.522;
   DATA[224,36] := 1.746067;
   DATA[224,37] := 190.0634;
   DATA[224,38] := 0.000128152;
   DATA[224,39] := 1.0;
   DATA[225,0] := 2.561573;
   DATA[225,1] := 525.9869;
   DATA[225,2] := 2.0;
   DATA[225,3] := 2.0;
   DATA[225,4] := 262.0802;
   DATA[225,5] := 8.391951;
   DATA[225,6] := 328.2748;
   DATA[225,7] := 2.440265;
   DATA[225,8] := 2.0;
   DATA[225,9] := 2.0;
   DATA[225,10] := 2.0;
   DATA[225,11] := 19.75479;
   DATA[225,12] := 2.210037;
   DATA[225,13] := 966.7393;
   DATA[225,14] := 1.0;
   DATA[225,15] := 2.0;
   DATA[225,16] := 1.0;
   DATA[225,17] := 1.0;
   DATA[225,18] := 1.0;
   DATA[225,19] := 2.0;
   DATA[225,20] := 148.808;
   DATA[225,21] := 155.7806;
   DATA[225,22] := 1.720565;
   DATA[225,23] := 959.4463;
   DATA[225,24] := 2.0;
   DATA[225,25] := 2.0;
   DATA[225,26] := 7.876058;
   DATA[225,27] := 144.7065;
   DATA[225,28] := 264.131;
   DATA[225,29] := 12.07383;
   DATA[225,30] := 1.731095;
   DATA[225,31] := 1.312284;
   DATA[225,32] := 0.7353967;
   DATA[225,33] := 0.3084905;
   DATA[225,34] := 2.0;
   DATA[225,35] := 251.522;
   DATA[225,36] := 1.746067;
   DATA[225,37] := 190.0795;
   DATA[225,38] := 0.000128152;
   DATA[225,39] := 1.0;
   DATA[226,0] := 2.549082;
   DATA[226,1] := 525.83;
   DATA[226,2] := 2.0;
   DATA[226,3] := 2.0;
   DATA[226,4] := 262.0802;
   DATA[226,5] := 8.391951;
   DATA[226,6] := 328.2748;
   DATA[226,7] := 2.440265;
   DATA[226,8] := 2.0;
   DATA[226,9] := 2.0;
   DATA[226,10] := 2.0;
   DATA[226,11] := 19.76439;
   DATA[226,12] := 2.210037;
   DATA[226,13] := 966.3388;
   DATA[226,14] := 1.0;
   DATA[226,15] := 2.0;
   DATA[226,16] := 1.0;
   DATA[226,17] := 1.0;
   DATA[226,18] := 1.0;
   DATA[226,19] := 2.0;
   DATA[226,20] := 148.808;
   DATA[226,21] := 155.7806;
   DATA[226,22] := 1.720565;
   DATA[226,23] := 959.9077;
   DATA[226,24] := 2.0;
   DATA[226,25] := 2.0;
   DATA[226,26] := 7.876058;
   DATA[226,27] := 144.7065;
   DATA[226,28] := 264.131;
   DATA[226,29] := 12.07383;
   DATA[226,30] := 1.731095;
   DATA[226,31] := 1.302805;
   DATA[226,32] := 0.7353967;
   DATA[226,33] := 0.3084905;
   DATA[226,34] := 2.0;
   DATA[226,35] := 251.522;
   DATA[226,36] := 1.746067;
   DATA[226,37] := 190.1596;
   DATA[226,38] := 0.000128152;
   DATA[226,39] := 1.0;
   DATA[227,0] := 2.530827;
   DATA[227,1] := 525.83;
   DATA[227,2] := 2.0;
   DATA[227,3] := 2.0;
   DATA[227,4] := 262.0802;
   DATA[227,5] := 8.391951;
   DATA[227,6] := 328.2748;
   DATA[227,7] := 2.441162;
   DATA[227,8] := 2.0;
   DATA[227,9] := 2.0;
   DATA[227,10] := 2.0;
   DATA[227,11] := 19.7836;
   DATA[227,12] := 2.210037;
   DATA[227,13] := 966.0184;
   DATA[227,14] := 1.0;
   DATA[227,15] := 2.0;
   DATA[227,16] := 1.0;
   DATA[227,17] := 1.0;
   DATA[227,18] := 1.0;
   DATA[227,19] := 2.0;
   DATA[227,20] := 148.808;
   DATA[227,21] := 155.7806;
   DATA[227,22] := 1.720565;
   DATA[227,23] := 960.5614;
   DATA[227,24] := 2.0;
   DATA[227,25] := 2.0;
   DATA[227,26] := 7.876058;
   DATA[227,27] := 144.7065;
   DATA[227,28] := 264.0989;
   DATA[227,29] := 12.07383;
   DATA[227,30] := 1.731095;
   DATA[227,31] := 1.298194;
   DATA[227,32] := 0.7361649;
   DATA[227,33] := 0.3084905;
   DATA[227,34] := 2.0;
   DATA[227,35] := 251.522;
   DATA[227,36] := 1.746067;
   DATA[227,37] := 190.1596;
   DATA[227,38] := 0.000128152;
   DATA[227,39] := 1.0;
   DATA[228,0] := 2.510009;
   DATA[228,1] := 526.0262;
   DATA[228,2] := 2.0;
   DATA[228,3] := 2.0;
   DATA[228,4] := 262.0802;
   DATA[228,5] := 8.391951;
   DATA[228,6] := 328.2748;
   DATA[228,7] := 2.441547;
   DATA[228,8] := 2.0;
   DATA[228,9] := 2.0;
   DATA[228,10] := 2.0;
   DATA[228,11] := 19.73238;
   DATA[228,12] := 2.211575;
   DATA[228,13] := 965.9382;
   DATA[228,14] := 1.0;
   DATA[228,15] := 2.0;
   DATA[228,16] := 1.0;
   DATA[228,17] := 1.0;
   DATA[228,18] := 1.0;
   DATA[228,19] := 2.0;
   DATA[228,20] := 148.808;
   DATA[228,21] := 155.7806;
   DATA[228,22] := 1.720565;
   DATA[228,23] := 960.7537;
   DATA[228,24] := 2.0;
   DATA[228,25] := 2.0;
   DATA[228,26] := 7.876058;
   DATA[228,27] := 144.7065;
   DATA[228,28] := 264.0989;
   DATA[228,29] := 12.07383;
   DATA[228,30] := 1.731095;
   DATA[228,31] := 1.282823;
   DATA[228,32] := 0.7384694;
   DATA[228,33] := 0.3084905;
   DATA[228,34] := 2.0;
   DATA[228,35] := 251.522;
   DATA[228,36] := 1.746067;
   DATA[228,37] := 190.1596;
   DATA[228,38] := 0.000128152;
   DATA[228,39] := 1.0;
   DATA[229,0] := 2.492073;
   DATA[229,1] := 526.0262;
   DATA[229,2] := 2.0;
   DATA[229,3] := 2.0;
   DATA[229,4] := 262.0802;
   DATA[229,5] := 8.391951;
   DATA[229,6] := 328.2748;
   DATA[229,7] := 2.441547;
   DATA[229,8] := 2.0;
   DATA[229,9] := 2.0;
   DATA[229,10] := 2.0;
   DATA[229,11] := 19.72598;
   DATA[229,12] := 2.213496;
   DATA[229,13] := 966.1786;
   DATA[229,14] := 1.0;
   DATA[229,15] := 2.0;
   DATA[229,16] := 1.0;
   DATA[229,17] := 1.0;
   DATA[229,18] := 1.0;
   DATA[229,19] := 2.0;
   DATA[229,20] := 148.808;
   DATA[229,21] := 155.7806;
   DATA[229,22] := 1.719156;
   DATA[229,23] := 960.7921;
   DATA[229,24] := 2.0;
   DATA[229,25] := 2.0;
   DATA[229,26] := 7.876058;
   DATA[229,27] := 144.7065;
   DATA[229,28] := 264.0989;
   DATA[229,29] := 12.07383;
   DATA[229,30] := 1.731095;
   DATA[229,31] := 1.282183;
   DATA[229,32] := 0.7353967;
   DATA[229,33] := 0.3084265;
   DATA[229,34] := 2.0;
   DATA[229,35] := 251.522;
   DATA[229,36] := 1.746067;
   DATA[229,37] := 190.1596;
   DATA[229,38] := 0.000128152;
   DATA[229,39] := 1.0;
   DATA[230,0] := 2.471255;
   DATA[230,1] := 526.1832;
   DATA[230,2] := 2.0;
   DATA[230,3] := 2.0;
   DATA[230,4] := 262.0802;
   DATA[230,5] := 8.391951;
   DATA[230,6] := 328.2748;
   DATA[230,7] := 2.441547;
   DATA[230,8] := 2.0;
   DATA[230,9] := 2.0;
   DATA[230,10] := 2.0;
   DATA[230,11] := 19.72598;
   DATA[230,12] := 2.213496;
   DATA[230,13] := 966.2587;
   DATA[230,14] := 1.0;
   DATA[230,15] := 2.0;
   DATA[230,16] := 1.0;
   DATA[230,17] := 1.0;
   DATA[230,18] := 1.0;
   DATA[230,19] := 2.0;
   DATA[230,20] := 148.808;
   DATA[230,21] := 155.7806;
   DATA[230,22] := 1.719156;
   DATA[230,23] := 961.1766;
   DATA[230,24] := 2.0;
   DATA[230,25] := 2.0;
   DATA[230,26] := 7.876058;
   DATA[230,27] := 144.8603;
   DATA[230,28] := 264.0989;
   DATA[230,29] := 12.07383;
   DATA[230,30] := 1.733017;
   DATA[230,31] := 1.28705;
   DATA[230,32] := 0.7353967;
   DATA[230,33] := 0.3064407;
   DATA[230,34] := 2.0;
   DATA[230,35] := 251.522;
   DATA[230,36] := 1.746067;
   DATA[230,37] := 190.1596;
   DATA[230,38] := 0.000128152;
   DATA[230,39] := 1.0;
   DATA[231,0] := 2.452359;
   DATA[231,1] := 526.4188;
   DATA[231,2] := 2.0;
   DATA[231,3] := 2.0;
   DATA[231,4] := 262.0802;
   DATA[231,5] := 8.391951;
   DATA[231,6] := 328.2748;
   DATA[231,7] := 2.4427;
   DATA[231,8] := 2.0;
   DATA[231,9] := 2.0;
   DATA[231,10] := 2.0;
   DATA[231,11] := 19.72598;
   DATA[231,12] := 2.21119;
   DATA[231,13] := 966.1786;
   DATA[231,14] := 1.0;
   DATA[231,15] := 2.0;
   DATA[231,16] := 1.0;
   DATA[231,17] := 1.0;
   DATA[231,18] := 1.0;
   DATA[231,19] := 2.0;
   DATA[231,20] := 148.808;
   DATA[231,21] := 155.7806;
   DATA[231,22] := 1.719156;
   DATA[231,23] := 961.1382;
   DATA[231,24] := 2.0;
   DATA[231,25] := 2.0;
   DATA[231,26] := 7.876058;
   DATA[231,27] := 144.8603;
   DATA[231,28] := 264.0989;
   DATA[231,29] := 12.07383;
   DATA[231,30] := 1.733914;
   DATA[231,31] := 1.279877;
   DATA[231,32] := 0.7353967;
   DATA[231,33] := 0.3064407;
   DATA[231,34] := 2.0;
   DATA[231,35] := 251.522;
   DATA[231,36] := 1.746067;
   DATA[231,37] := 190.1596;
   DATA[231,38] := 0.000128152;
   DATA[231,39] := 1.0;
   DATA[232,0] := 2.436345;
   DATA[232,1] := 526.2617;
   DATA[232,2] := 2.0;
   DATA[232,3] := 2.0;
   DATA[232,4] := 262.0802;
   DATA[232,5] := 8.391951;
   DATA[232,6] := 328.2748;
   DATA[232,7] := 2.442828;
   DATA[232,8] := 2.0;
   DATA[232,9] := 2.0;
   DATA[232,10] := 2.0;
   DATA[232,11] := 19.72598;
   DATA[232,12] := 2.21119;
   DATA[232,13] := 966.0184;
   DATA[232,14] := 1.0;
   DATA[232,15] := 2.0;
   DATA[232,16] := 1.0;
   DATA[232,17] := 1.0;
   DATA[232,18] := 1.0;
   DATA[232,19] := 2.0;
   DATA[232,20] := 148.808;
   DATA[232,21] := 155.7806;
   DATA[232,22] := 1.720053;
   DATA[232,23] := 961.292;
   DATA[232,24] := 2.0;
   DATA[232,25] := 2.0;
   DATA[232,26] := 7.876058;
   DATA[232,27] := 144.8603;
   DATA[232,28] := 264.0989;
   DATA[232,29] := 12.07383;
   DATA[232,30] := 1.733914;
   DATA[232,31] := 1.281286;
   DATA[232,32] := 0.7353967;
   DATA[232,33] := 0.3064407;
   DATA[232,34] := 2.0;
   DATA[232,35] := 251.522;
   DATA[232,36] := 1.617916;
   DATA[232,37] := 190.1596;
   DATA[232,38] := 0.000128152;
   DATA[232,39] := 1.0;
   DATA[233,0] := 2.43026;
   DATA[233,1] := 526.0655;
   DATA[233,2] := 2.0;
   DATA[233,3] := 2.0;
   DATA[233,4] := 262.0802;
   DATA[233,5] := 8.391951;
   DATA[233,6] := 328.2748;
   DATA[233,7] := 2.444238;
   DATA[233,8] := 2.0;
   DATA[233,9] := 2.0;
   DATA[233,10] := 2.0;
   DATA[233,11] := 19.70037;
   DATA[233,12] := 2.21119;
   DATA[233,13] := 966.5391;
   DATA[233,14] := 1.0;
   DATA[233,15] := 2.0;
   DATA[233,16] := 1.0;
   DATA[233,17] := 1.0;
   DATA[233,18] := 1.0;
   DATA[233,19] := 2.0;
   DATA[233,20] := 148.808;
   DATA[233,21] := 155.7806;
   DATA[233,22] := 1.722359;
   DATA[233,23] := 961.6381;
   DATA[233,24] := 2.0;
   DATA[233,25] := 2.0;
   DATA[233,26] := 7.876058;
   DATA[233,27] := 144.8603;
   DATA[233,28] := 264.0989;
   DATA[233,29] := 12.07383;
   DATA[233,30] := 1.731479;
   DATA[233,31] := 1.291918;
   DATA[233,32] := 0.7353967;
   DATA[233,33] := 0.3064407;
   DATA[233,34] := 2.0;
   DATA[233,35] := 251.522;
   DATA[233,36] := 1.617916;
   DATA[233,37] := 190.1596;
   DATA[233,38] := 0.000128152;
   DATA[233,39] := 1.0;
   DATA[234,0] := 2.428338;
   DATA[234,1] := 526.2617;
   DATA[234,2] := 2.0;
   DATA[234,3] := 2.0;
   DATA[234,4] := 262.0802;
   DATA[234,5] := 8.391951;
   DATA[234,6] := 328.2748;
   DATA[234,7] := 2.445007;
   DATA[234,8] := 2.0;
   DATA[234,9] := 2.0;
   DATA[234,10] := 2.0;
   DATA[234,11] := 19.70037;
   DATA[234,12] := 2.21119;
   DATA[234,13] := 966.4189;
   DATA[234,14] := 1.0;
   DATA[234,15] := 2.0;
   DATA[234,16] := 1.0;
   DATA[234,17] := 1.0;
   DATA[234,18] := 1.0;
   DATA[234,19] := 2.0;
   DATA[234,20] := 148.808;
   DATA[234,21] := 155.9087;
   DATA[234,22] := 1.722359;
   DATA[234,23] := 961.4458;
   DATA[234,24] := 2.0;
   DATA[234,25] := 2.0;
   DATA[234,26] := 7.876058;
   DATA[234,27] := 144.8603;
   DATA[234,28] := 264.0989;
   DATA[234,29] := 12.07383;
   DATA[234,30] := 1.731095;
   DATA[234,31] := 1.297169;
   DATA[234,32] := 0.7353967;
   DATA[234,33] := 0.3064407;
   DATA[234,34] := 2.0;
   DATA[234,35] := 251.522;
   DATA[234,36] := 1.617916;
   DATA[234,37] := 190.1596;
   DATA[234,38] := 0.000128152;
   DATA[234,39] := 1.0;
   DATA[235,0] := 2.438587;
   DATA[235,1] := 525.9084;
   DATA[235,2] := 2.0;
   DATA[235,3] := 2.0;
   DATA[235,4] := 262.0802;
   DATA[235,5] := 8.391951;
   DATA[235,6] := 328.2748;
   DATA[235,7] := 2.445007;
   DATA[235,8] := 2.0;
   DATA[235,9] := 2.0;
   DATA[235,10] := 2.0;
   DATA[235,11] := 19.70037;
   DATA[235,12] := 2.210037;
   DATA[235,13] := 966.5791;
   DATA[235,14] := 1.0;
   DATA[235,15] := 2.0;
   DATA[235,16] := 1.0;
   DATA[235,17] := 1.0;
   DATA[235,18] := 1.0;
   DATA[235,19] := 2.0;
   DATA[235,20] := 148.808;
   DATA[235,21] := 155.9087;
   DATA[235,22] := 1.722359;
   DATA[235,23] := 961.5612;
   DATA[235,24] := 2.0;
   DATA[235,25] := 2.0;
   DATA[235,26] := 7.876058;
   DATA[235,27] := 144.8603;
   DATA[235,28] := 264.0989;
   DATA[235,29] := 12.07383;
   DATA[235,30] := 1.731095;
   DATA[235,31] := 1.308825;
   DATA[235,32] := 0.7353967;
   DATA[235,33] := 0.3064407;
   DATA[235,34] := 2.0;
   DATA[235,35] := 251.522;
   DATA[235,36] := 1.617916;
   DATA[235,37] := 190.1596;
   DATA[235,38] := 0.000128152;
   DATA[235,39] := 1.0;
   DATA[236,0] := 2.48791;
   DATA[236,1] := 525.4767;
   DATA[236,2] := 2.0;
   DATA[236,3] := 2.0;
   DATA[236,4] := 262.0802;
   DATA[236,5] := 8.391951;
   DATA[236,6] := 328.2748;
   DATA[236,7] := 2.445007;
   DATA[236,8] := 2.0;
   DATA[236,9] := 2.0;
   DATA[236,10] := 2.0;
   DATA[236,11] := 19.70037;
   DATA[236,12] := 2.210037;
   DATA[236,13] := 966.8595;
   DATA[236,14] := 1.0;
   DATA[236,15] := 2.0;
   DATA[236,16] := 1.0;
   DATA[236,17] := 1.0;
   DATA[236,18] := 1.0;
   DATA[236,19] := 2.0;
   DATA[236,20] := 148.808;
   DATA[236,21] := 155.9087;
   DATA[236,22] := 1.722359;
   DATA[236,23] := 962.0226;
   DATA[236,24] := 2.0;
   DATA[236,25] := 2.0;
   DATA[236,26] := 7.876058;
   DATA[236,27] := 144.8603;
   DATA[236,28] := 264.0989;
   DATA[236,29] := 12.07383;
   DATA[236,30] := 1.731095;
   DATA[236,31] := 1.312028;
   DATA[236,32] := 0.7353967;
   DATA[236,33] := 0.3064407;
   DATA[236,34] := 2.0;
   DATA[236,35] := 251.522;
   DATA[236,36] := 1.617916;
   DATA[236,37] := 190.1596;
   DATA[236,38] := 0.000128152;
   DATA[236,39] := 1.0;
   DATA[237,0] := 2.536912;
   DATA[237,1] := 524.9271;
   DATA[237,2] := 2.0;
   DATA[237,3] := 2.0;
   DATA[237,4] := 262.0802;
   DATA[237,5] := 8.391951;
   DATA[237,6] := 328.2748;
   DATA[237,7] := 2.444623;
   DATA[237,8] := 2.0;
   DATA[237,9] := 2.0;
   DATA[237,10] := 2.0;
   DATA[237,11] := 19.75479;
   DATA[237,12] := 2.210037;
   DATA[237,13] := 966.7794;
   DATA[237,14] := 1.0;
   DATA[237,15] := 2.0;
   DATA[237,16] := 1.0;
   DATA[237,17] := 1.0;
   DATA[237,18] := 1.0;
   DATA[237,19] := 2.0;
   DATA[237,20] := 148.808;
   DATA[237,21] := 155.9087;
   DATA[237,22] := 1.722359;
   DATA[237,23] := 962.3302;
   DATA[237,24] := 2.0;
   DATA[237,25] := 2.0;
   DATA[237,26] := 7.876058;
   DATA[237,27] := 144.8603;
   DATA[237,28] := 264.0989;
   DATA[237,29] := 12.07383;
   DATA[237,30] := 1.731095;
   DATA[237,31] := 1.297169;
   DATA[237,32] := 0.7353967;
   DATA[237,33] := 0.3069532;
   DATA[237,34] := 2.0;
   DATA[237,35] := 251.522;
   DATA[237,36] := 1.617916;
   DATA[237,37] := 190.1596;
   DATA[237,38] := 0.000128152;
   DATA[237,39] := 1.0;
   DATA[238,0] := 2.582711;
   DATA[238,1] := 524.9271;
   DATA[238,2] := 2.0;
   DATA[238,3] := 2.0;
   DATA[238,4] := 262.0802;
   DATA[238,5] := 8.391951;
   DATA[238,6] := 328.2748;
   DATA[238,7] := 2.444238;
   DATA[238,8] := 2.0;
   DATA[238,9] := 2.0;
   DATA[238,10] := 2.0;
   DATA[238,11] := 19.7804;
   DATA[238,12] := 2.210037;
   DATA[238,13] := 967.3401;
   DATA[238,14] := 1.0;
   DATA[238,15] := 2.0;
   DATA[238,16] := 1.0;
   DATA[238,17] := 1.0;
   DATA[238,18] := 1.0;
   DATA[238,19] := 2.0;
   DATA[238,20] := 148.808;
   DATA[238,21] := 155.9087;
   DATA[238,22] := 1.720565;
   DATA[238,23] := 962.3302;
   DATA[238,24] := 2.0;
   DATA[238,25] := 2.0;
   DATA[238,26] := 7.876058;
   DATA[238,27] := 144.8603;
   DATA[238,28] := 264.0989;
   DATA[238,29] := 12.07383;
   DATA[238,30] := 1.731095;
   DATA[238,31] := 1.283592;
   DATA[238,32] := 0.7353967;
   DATA[238,33] := 0.3069532;
   DATA[238,34] := 2.0;
   DATA[238,35] := 251.522;
   DATA[238,36] := 1.746067;
   DATA[238,37] := 190.1596;
   DATA[238,38] := 0.000128152;
   DATA[238,39] := 1.0;
   DATA[239,0] := 2.614739;
   DATA[239,1] := 525.2411;
   DATA[239,2] := 2.0;
   DATA[239,3] := 2.0;
   DATA[239,4] := 262.0802;
   DATA[239,5] := 8.391951;
   DATA[239,6] := 328.2748;
   DATA[239,7] := 2.441547;
   DATA[239,8] := 2.0;
   DATA[239,9] := 2.0;
   DATA[239,10] := 2.0;
   DATA[239,11] := 19.7804;
   DATA[239,12] := 2.210037;
   DATA[239,13] := 967.6606;
   DATA[239,14] := 1.0;
   DATA[239,15] := 2.0;
   DATA[239,16] := 1.0;
   DATA[239,17] := 1.0;
   DATA[239,18] := 1.0;
   DATA[239,19] := 2.0;
   DATA[239,20] := 148.808;
   DATA[239,21] := 155.9087;
   DATA[239,22] := 1.720565;
   DATA[239,23] := 962.1379;
   DATA[239,24] := 2.0;
   DATA[239,25] := 2.0;
   DATA[239,26] := 7.876058;
   DATA[239,27] := 144.8603;
   DATA[239,28] := 263.9067;
   DATA[239,29] := 12.07383;
   DATA[239,30] := 1.728916;
   DATA[239,31] := 1.281542;
   DATA[239,32] := 0.7353967;
   DATA[239,33] := 0.3069532;
   DATA[239,34] := 2.0;
   DATA[239,35] := 251.522;
   DATA[239,36] := 1.746067;
   DATA[239,37] := 190.1596;
   DATA[239,38] := 0.000128152;
   DATA[239,39] := 1.0;
   DATA[240,0] := 2.653813;
   DATA[240,1] := 525.8692;
   DATA[240,2] := 2.0;
   DATA[240,3] := 2.0;
   DATA[240,4] := 262.0802;
   DATA[240,5] := 8.39131;
   DATA[240,6] := 328.2748;
   DATA[240,7] := 2.440521;
   DATA[240,8] := 2.0;
   DATA[240,9] := 2.0;
   DATA[240,10] := 2.0;
   DATA[240,11] := 19.7804;
   DATA[240,12] := 2.210037;
   DATA[240,13] := 967.9409;
   DATA[240,14] := 1.0;
   DATA[240,15] := 2.0;
   DATA[240,16] := 1.0;
   DATA[240,17] := 1.0;
   DATA[240,18] := 1.0;
   DATA[240,19] := 2.0;
   DATA[240,20] := 148.808;
   DATA[240,21] := 155.9087;
   DATA[240,22] := 1.720565;
   DATA[240,23] := 962.4071;
   DATA[240,24] := 2.0;
   DATA[240,25] := 2.0;
   DATA[240,26] := 7.876058;
   DATA[240,27] := 144.8603;
   DATA[240,28] := 263.9067;
   DATA[240,29] := 12.07383;
   DATA[240,30] := 1.728531;
   DATA[240,31] := 1.286794;
   DATA[240,32] := 0.7353967;
   DATA[240,33] := 0.3069532;
   DATA[240,34] := 2.0;
   DATA[240,35] := 251.522;
   DATA[240,36] := 1.746067;
   DATA[240,37] := 190.1596;
   DATA[240,38] := 0.000128152;
   DATA[240,39] := 1.0;
   DATA[241,0] := 2.671428;
   DATA[241,1] := 526.458;
   DATA[241,2] := 2.0;
   DATA[241,3] := 2.0;
   DATA[241,4] := 262.0802;
   DATA[241,5] := 8.388746;
   DATA[241,6] := 328.2748;
   DATA[241,7] := 2.440521;
   DATA[241,8] := 2.0;
   DATA[241,9] := 2.0;
   DATA[241,10] := 2.0;
   DATA[241,11] := 19.7804;
   DATA[241,12] := 2.210037;
   DATA[241,13] := 968.0611;
   DATA[241,14] := 1.0;
   DATA[241,15] := 2.0;
   DATA[241,16] := 1.0;
   DATA[241,17] := 1.0;
   DATA[241,18] := 1.0;
   DATA[241,19] := 2.0;
   DATA[241,20] := 148.808;
   DATA[241,21] := 155.9087;
   DATA[241,22] := 1.722359;
   DATA[241,23] := 962.3302;
   DATA[241,24] := 2.0;
   DATA[241,25] := 2.0;
   DATA[241,26] := 7.876058;
   DATA[241,27] := 144.8603;
   DATA[241,28] := 263.9067;
   DATA[241,29] := 12.07383;
   DATA[241,30] := 1.728531;
   DATA[241,31] := 1.285641;
   DATA[241,32] := 0.7353967;
   DATA[241,33] := 0.3064407;
   DATA[241,34] := 2.0;
   DATA[241,35] := 251.522;
   DATA[241,36] := 1.649953;
   DATA[241,37] := 190.1596;
   DATA[241,38] := 0.000128152;
   DATA[241,39] := 1.0;
   DATA[242,0] := 2.675592;
   DATA[242,1] := 526.615;
   DATA[242,2] := 2.0;
   DATA[242,3] := 2.0;
   DATA[242,4] := 262.0802;
   DATA[242,5] := 8.388746;
   DATA[242,6] := 328.2748;
   DATA[242,7] := 2.440521;
   DATA[242,8] := 2.0;
   DATA[242,9] := 2.0;
   DATA[242,10] := 2.0;
   DATA[242,11] := 19.75159;
   DATA[242,12] := 2.211959;
   DATA[242,13] := 968.2213;
   DATA[242,14] := 1.0;
   DATA[242,15] := 2.0;
   DATA[242,16] := 1.0;
   DATA[242,17] := 1.0;
   DATA[242,18] := 1.0;
   DATA[242,19] := 2.0;
   DATA[242,20] := 148.808;
   DATA[242,21] := 155.9087;
   DATA[242,22] := 1.722359;
   DATA[242,23] := 962.2533;
   DATA[242,24] := 2.0;
   DATA[242,25] := 2.0;
   DATA[242,26] := 7.876058;
   DATA[242,27] := 144.8603;
   DATA[242,28] := 263.9067;
   DATA[242,29] := 12.07383;
   DATA[242,30] := 1.728531;
   DATA[242,31] := 1.299475;
   DATA[242,32] := 0.7353967;
   DATA[242,33] := 0.3064407;
   DATA[242,34] := 2.0;
   DATA[242,35] := 251.522;
   DATA[242,36] := 1.649953;
   DATA[242,37] := 190.1596;
   DATA[242,38] := 0.000128152;
   DATA[242,39] := 1.0;
   DATA[243,0] := 2.649329;
   DATA[243,1] := 526.9683;
   DATA[243,2] := 2.0;
   DATA[243,3] := 2.0;
   DATA[243,4] := 262.0802;
   DATA[243,5] := 8.388746;
   DATA[243,6] := 328.2748;
   DATA[243,7] := 2.440521;
   DATA[243,8] := 2.0;
   DATA[243,9] := 2.0;
   DATA[243,10] := 2.0;
   DATA[243,11] := 19.69076;
   DATA[243,12] := 2.213496;
   DATA[243,13] := 968.2614;
   DATA[243,14] := 1.0;
   DATA[243,15] := 2.0;
   DATA[243,16] := 1.0;
   DATA[243,17] := 1.0;
   DATA[243,18] := 1.0;
   DATA[243,19] := 2.0;
   DATA[243,20] := 148.808;
   DATA[243,21] := 155.9087;
   DATA[243,22] := 1.722359;
   DATA[243,23] := 962.6378;
   DATA[243,24] := 2.0;
   DATA[243,25] := 2.0;
   DATA[243,26] := 7.876058;
   DATA[243,27] := 144.8603;
   DATA[243,28] := 263.9067;
   DATA[243,29] := 12.07383;
   DATA[243,30] := 1.73071;
   DATA[243,31] := 1.299475;
   DATA[243,32] := 0.7353967;
   DATA[243,33] := 0.3064407;
   DATA[243,34] := 2.0;
   DATA[243,35] := 251.4419;
   DATA[243,36] := 1.649953;
   DATA[243,37] := 190.1596;
   DATA[243,38] := 0.000128152;
   DATA[243,39] := 1.0;
   DATA[244,0] := 2.625628;
   DATA[244,1] := 527.3608;
   DATA[244,2] := 2.0;
   DATA[244,3] := 2.0;
   DATA[244,4] := 262.0802;
   DATA[244,5] := 8.388746;
   DATA[244,6] := 328.2748;
   DATA[244,7] := 2.440137;
   DATA[244,8] := 2.0;
   DATA[244,9] := 2.0;
   DATA[244,10] := 2.0;
   DATA[244,11] := 19.65235;
   DATA[244,12] := 2.213496;
   DATA[244,13] := 968.6218;
   DATA[244,14] := 1.0;
   DATA[244,15] := 2.0;
   DATA[244,16] := 1.0;
   DATA[244,17] := 1.0;
   DATA[244,18] := 1.0;
   DATA[244,19] := 2.0;
   DATA[244,20] := 148.808;
   DATA[244,21] := 155.9087;
   DATA[244,22] := 1.722359;
   DATA[244,23] := 963.0607;
   DATA[244,24] := 2.0;
   DATA[244,25] := 2.0;
   DATA[244,26] := 7.876058;
   DATA[244,27] := 144.8603;
   DATA[244,28] := 263.9067;
   DATA[244,29] := 12.07383;
   DATA[244,30] := 1.731351;
   DATA[244,31] := 1.282823;
   DATA[244,32] := 0.7353967;
   DATA[244,33] := 0.3064407;
   DATA[244,34] := 2.0;
   DATA[244,35] := 251.4419;
   DATA[244,36] := 1.649953;
   DATA[244,37] := 190.1596;
   DATA[244,38] := 0.000128152;
   DATA[244,39] := 1.0;
   DATA[245,0] := 2.620824;
   DATA[245,1] := 527.6356;
   DATA[245,2] := 2.0;
   DATA[245,3] := 2.0;
   DATA[245,4] := 262.0802;
   DATA[245,5] := 8.39131;
   DATA[245,6] := 328.2748;
   DATA[245,7] := 2.440137;
   DATA[245,8] := 2.0;
   DATA[245,9] := 2.0;
   DATA[245,10] := 2.0;
   DATA[245,11] := 19.65235;
   DATA[245,12] := 2.213368;
   DATA[245,13] := 968.3815;
   DATA[245,14] := 1.0;
   DATA[245,15] := 2.0;
   DATA[245,16] := 1.0;
   DATA[245,17] := 1.0;
   DATA[245,18] := 1.0;
   DATA[245,19] := 2.0;
   DATA[245,20] := 148.808;
   DATA[245,21] := 155.9087;
   DATA[245,22] := 1.722359;
   DATA[245,23] := 962.9069;
   DATA[245,24] := 2.0;
   DATA[245,25] := 2.0;
   DATA[245,26] := 7.876058;
   DATA[245,27] := 144.8603;
   DATA[245,28] := 263.9067;
   DATA[245,29] := 12.07383;
   DATA[245,30] := 1.731479;
   DATA[245,31] := 1.27232;
   DATA[245,32] := 0.7353967;
   DATA[245,33] := 0.3064407;
   DATA[245,34] := 2.0;
   DATA[245,35] := 251.4419;
   DATA[245,36] := 1.826162;
   DATA[245,37] := 190.3679;
   DATA[245,38] := 0.000128152;
   DATA[245,39] := 1.0;
   DATA[246,0] := 2.620504;
   DATA[246,1] := 528.0674;
   DATA[246,2] := 2.0;
   DATA[246,3] := 2.0;
   DATA[246,4] := 262.0802;
   DATA[246,5] := 8.39131;
   DATA[246,6] := 328.2748;
   DATA[246,7] := 2.440137;
   DATA[246,8] := 2.0;
   DATA[246,9] := 2.0;
   DATA[246,10] := 2.0;
   DATA[246,11] := 19.62674;
   DATA[246,12] := 2.211575;
   DATA[246,13] := 968.5818;
   DATA[246,14] := 1.0;
   DATA[246,15] := 2.0;
   DATA[246,16] := 1.0;
   DATA[246,17] := 1.0;
   DATA[246,18] := 1.0;
   DATA[246,19] := 2.0;
   DATA[246,20] := 148.808;
   DATA[246,21] := 155.9087;
   DATA[246,22] := 1.722359;
   DATA[246,23] := 962.8685;
   DATA[246,24] := 2.0;
   DATA[246,25] := 2.0;
   DATA[246,26] := 7.876058;
   DATA[246,27] := 144.8603;
   DATA[246,28] := 263.9387;
   DATA[246,29] := 12.07383;
   DATA[246,30] := 1.731479;
   DATA[246,31] := 1.262329;
   DATA[246,32] := 0.7353967;
   DATA[246,33] := 0.3064407;
   DATA[246,34] := 2.0;
   DATA[246,35] := 251.4419;
   DATA[246,36] := 1.826162;
   DATA[246,37] := 190.3679;
   DATA[246,38] := 0.000128152;
   DATA[246,39] := 1.0;
   DATA[247,0] := 2.608334;
   DATA[247,1] := 528.2636;
   DATA[247,2] := 2.0;
   DATA[247,3] := 2.0;
   DATA[247,4] := 262.0802;
   DATA[247,5] := 8.39131;
   DATA[247,6] := 328.2748;
   DATA[247,7] := 2.441675;
   DATA[247,8] := 2.0;
   DATA[247,9] := 2.0;
   DATA[247,10] := 2.0;
   DATA[247,11] := 19.62674;
   DATA[247,12] := 2.209397;
   DATA[247,13] := 968.9824;
   DATA[247,14] := 1.0;
   DATA[247,15] := 2.0;
   DATA[247,16] := 1.0;
   DATA[247,17] := 1.0;
   DATA[247,18] := 1.0;
   DATA[247,19] := 2.0;
   DATA[247,20] := 148.808;
   DATA[247,21] := 155.9087;
   DATA[247,22] := 1.722359;
   DATA[247,23] := 963.0607;
   DATA[247,24] := 2.0;
   DATA[247,25] := 2.0;
   DATA[247,26] := 7.876058;
   DATA[247,27] := 144.9116;
   DATA[247,28] := 264.0989;
   DATA[247,29] := 12.07383;
   DATA[247,30] := 1.731479;
   DATA[247,31] := 1.261432;
   DATA[247,32] := 0.7353967;
   DATA[247,33] := 0.3064407;
   DATA[247,34] := 2.0;
   DATA[247,35] := 251.4419;
   DATA[247,36] := 1.762086;
   DATA[247,37] := 190.2397;
   DATA[247,38] := 0.000128152;
   DATA[247,39] := 1.0;
   DATA[248,0] := 2.583992;
   DATA[248,1] := 528.0281;
   DATA[248,2] := 2.0;
   DATA[248,3] := 2.0;
   DATA[248,4] := 262.0802;
   DATA[248,5] := 8.39131;
   DATA[248,6] := 328.2748;
   DATA[248,7] := 2.442188;
   DATA[248,8] := 2.0;
   DATA[248,9] := 2.0;
   DATA[248,10] := 2.0;
   DATA[248,11] := 19.62674;
   DATA[248,12] := 2.209397;
   DATA[248,13] := 969.1426;
   DATA[248,14] := 1.0;
   DATA[248,15] := 2.0;
   DATA[248,16] := 1.0;
   DATA[248,17] := 1.0;
   DATA[248,18] := 1.0;
   DATA[248,19] := 2.0;
   DATA[248,20] := 148.808;
   DATA[248,21] := 155.9087;
   DATA[248,22] := 1.722359;
   DATA[248,23] := 962.8685;
   DATA[248,24] := 2.0;
   DATA[248,25] := 2.0;
   DATA[248,26] := 7.876058;
   DATA[248,27] := 144.9885;
   DATA[248,28] := 264.0989;
   DATA[248,29] := 12.15073;
   DATA[248,30] := 1.731479;
   DATA[248,31] := 1.279365;
   DATA[248,32] := 0.7353967;
   DATA[248,33] := 0.3064407;
   DATA[248,34] := 2.0;
   DATA[248,35] := 251.4419;
   DATA[248,36] := 1.69801;
   DATA[248,37] := 190.0795;
   DATA[248,38] := 0.000128152;
   DATA[248,39] := 1.0;
   DATA[249,0] := 2.571182;
   DATA[249,1] := 527.8711;
   DATA[249,2] := 2.0;
   DATA[249,3] := 2.0;
   DATA[249,4] := 262.0802;
   DATA[249,5] := 8.39131;
   DATA[249,6] := 328.2748;
   DATA[249,7] := 2.442188;
   DATA[249,8] := 2.0;
   DATA[249,9] := 2.0;
   DATA[249,10] := 2.0;
   DATA[249,11] := 19.65555;
   DATA[249,12] := 2.212728;
   DATA[249,13] := 969.1826;
   DATA[249,14] := 1.0;
   DATA[249,15] := 2.0;
   DATA[249,16] := 1.0;
   DATA[249,17] := 1.0;
   DATA[249,18] := 1.0;
   DATA[249,19] := 2.0;
   DATA[249,20] := 148.808;
   DATA[249,21] := 155.9087;
   DATA[249,22] := 1.718387;
   DATA[249,23] := 962.6762;
   DATA[249,24] := 2.0;
   DATA[249,25] := 2.0;
   DATA[249,26] := 7.876058;
   DATA[249,27] := 144.9885;
   DATA[249,28] := 264.0989;
   DATA[249,29] := 12.15073;
   DATA[249,30] := 1.730454;
   DATA[249,31] := 1.281542;
   DATA[249,32] := 0.7353967;
   DATA[249,33] := 0.3064407;
   DATA[249,34] := 2.0;
   DATA[249,35] := 251.4419;
   DATA[249,36] := 1.649953;
   DATA[249,37] := 190.0795;
   DATA[249,38] := 0.000128152;
   DATA[249,39] := 1.0;
   DATA[250,0] := 2.548762;
   DATA[250,1] := 527.8318;
   DATA[250,2] := 2.0;
   DATA[250,3] := 2.0;
   DATA[250,4] := 262.0802;
   DATA[250,5] := 8.39131;
   DATA[250,6] := 328.3004;
   DATA[250,7] := 2.442188;
   DATA[250,8] := 2.0;
   DATA[250,9] := 2.0;
   DATA[250,10] := 2.0;
   DATA[250,11] := 19.70037;
   DATA[250,12] := 2.212728;
   DATA[250,13] := 968.9824;
   DATA[250,14] := 1.0;
   DATA[250,15] := 2.0;
   DATA[250,16] := 1.0;
   DATA[250,17] := 1.0;
   DATA[250,18] := 1.0;
   DATA[250,19] := 2.0;
   DATA[250,20] := 148.808;
   DATA[250,21] := 155.9087;
   DATA[250,22] := 1.718387;
   DATA[250,23] := 962.5224;
   DATA[250,24] := 2.0;
   DATA[250,25] := 2.0;
   DATA[250,26] := 7.876058;
   DATA[250,27] := 144.9885;
   DATA[250,28] := 264.0989;
   DATA[250,29] := 12.15073;
   DATA[250,30] := 1.7293;
   DATA[250,31] := 1.290252;
   DATA[250,32] := 0.7353967;
   DATA[250,33] := 0.3064407;
   DATA[250,34] := 2.0;
   DATA[250,35] := 251.4419;
   DATA[250,36] := 1.649953;
   DATA[250,37] := 190.0154;
   DATA[250,38] := 0.000128152;
   DATA[250,39] := 1.0;
   DATA[251,0] := 2.535631;
   DATA[251,1] := 527.6356;
   DATA[251,2] := 2.0;
   DATA[251,3] := 2.0;
   DATA[251,4] := 262.0802;
   DATA[251,5] := 8.39131;
   DATA[251,6] := 328.3004;
   DATA[251,7] := 2.443469;
   DATA[251,8] := 2.0;
   DATA[251,9] := 2.0;
   DATA[251,10] := 2.0;
   DATA[251,11] := 19.70037;
   DATA[251,12] := 2.212728;
   DATA[251,13] := 968.8622;
   DATA[251,14] := 1.0;
   DATA[251,15] := 2.0;
   DATA[251,16] := 1.0;
   DATA[251,17] := 1.0;
   DATA[251,18] := 1.0;
   DATA[251,19] := 2.0;
   DATA[251,20] := 148.808;
   DATA[251,21] := 155.9087;
   DATA[251,22] := 1.718387;
   DATA[251,23] := 962.4456;
   DATA[251,24] := 2.0;
   DATA[251,25] := 2.0;
   DATA[251,26] := 7.876058;
   DATA[251,27] := 144.9885;
   DATA[251,28] := 264.0989;
   DATA[251,29] := 12.15073;
   DATA[251,30] := 1.7293;
   DATA[251,31] := 1.300243;
   DATA[251,32] := 0.7353967;
   DATA[251,33] := 0.3064407;
   DATA[251,34] := 2.0;
   DATA[251,35] := 251.1375;
   DATA[251,36] := 1.649953;
   DATA[251,37] := 189.8071;
   DATA[251,38] := 0.000128152;
   DATA[251,39] := 1.0;
   DATA[252,0] := 2.510329;
   DATA[252,1] := 527.7534;
   DATA[252,2] := 2.0;
   DATA[252,3] := 2.0;
   DATA[252,4] := 262.0802;
   DATA[252,5] := 8.39131;
   DATA[252,6] := 328.3004;
   DATA[252,7] := 2.443469;
   DATA[252,8] := 2.0;
   DATA[252,9] := 2.0;
   DATA[252,10] := 2.0;
   DATA[252,11] := 19.67796;
   DATA[252,12] := 2.210934;
   DATA[252,13] := 968.2213;
   DATA[252,14] := 1.0;
   DATA[252,15] := 2.0;
   DATA[252,16] := 1.0;
   DATA[252,17] := 1.0;
   DATA[252,18] := 1.0;
   DATA[252,19] := 2.0;
   DATA[252,20] := 148.808;
   DATA[252,21] := 155.9087;
   DATA[252,22] := 1.718387;
   DATA[252,23] := 962.4456;
   DATA[252,24] := 2.0;
   DATA[252,25] := 2.0;
   DATA[252,26] := 7.876058;
   DATA[252,27] := 144.9885;
   DATA[252,28] := 264.0989;
   DATA[252,29] := 12.15073;
   DATA[252,30] := 1.7293;
   DATA[252,31] := 1.302165;
   DATA[252,32] := 0.7353967;
   DATA[252,33] := 0.3064407;
   DATA[252,34] := 2.0;
   DATA[252,35] := 251.0574;
   DATA[252,36] := 1.649953;
   DATA[252,37] := 189.8071;
   DATA[252,38] := 0.000128152;
   DATA[252,39] := 1.0;
   DATA[253,0] := 2.502642;
   DATA[253,1] := 527.7534;
   DATA[253,2] := 2.0;
   DATA[253,3] := 2.0;
   DATA[253,4] := 262.0802;
   DATA[253,5] := 8.39131;
   DATA[253,6] := 328.3004;
   DATA[253,7] := 2.443469;
   DATA[253,8] := 2.0;
   DATA[253,9] := 2.0;
   DATA[253,10] := 2.0;
   DATA[253,11] := 19.66195;
   DATA[253,12] := 2.210934;
   DATA[253,13] := 967.7407;
   DATA[253,14] := 1.0;
   DATA[253,15] := 2.0;
   DATA[253,16] := 1.0;
   DATA[253,17] := 1.0;
   DATA[253,18] := 1.0;
   DATA[253,19] := 2.0;
   DATA[253,20] := 148.808;
   DATA[253,21] := 155.9087;
   DATA[253,22] := 1.718387;
   DATA[253,23] := 962.2148;
   DATA[253,24] := 2.0;
   DATA[253,25] := 2.0;
   DATA[253,26] := 7.876058;
   DATA[253,27] := 144.9885;
   DATA[253,28] := 264.0989;
   DATA[253,29] := 12.15073;
   DATA[253,30] := 1.7293;
   DATA[253,31] := 1.302165;
   DATA[253,32] := 0.7353967;
   DATA[253,33] := 0.3064407;
   DATA[253,34] := 2.0;
   DATA[253,35] := 250.8972;
   DATA[253,36] := 1.649953;
   DATA[253,37] := 189.8071;
   DATA[253,38] := 0.000128152;
   DATA[253,39] := 1.0;
   DATA[254,0] := 2.484707;
   DATA[254,1] := 528.4207;
   DATA[254,2] := 2.0;
   DATA[254,3] := 2.0;
   DATA[254,4] := 262.0802;
   DATA[254,5] := 8.39131;
   DATA[254,6] := 328.3004;
   DATA[254,7] := 2.443469;
   DATA[254,8] := 2.0;
   DATA[254,9] := 2.0;
   DATA[254,10] := 2.0;
   DATA[254,11] := 19.66195;
   DATA[254,12] := 2.210934;
   DATA[254,13] := 967.7407;
   DATA[254,14] := 1.0;
   DATA[254,15] := 2.0;
   DATA[254,16] := 1.0;
   DATA[254,17] := 1.0;
   DATA[254,18] := 1.0;
   DATA[254,19] := 2.0;
   DATA[254,20] := 148.808;
   DATA[254,21] := 155.9087;
   DATA[254,22] := 1.718387;
   DATA[254,23] := 962.5224;
   DATA[254,24] := 2.0;
   DATA[254,25] := 2.0;
   DATA[254,26] := 7.876058;
   DATA[254,27] := 144.9885;
   DATA[254,28] := 264.0989;
   DATA[254,29] := 12.15073;
   DATA[254,30] := 1.726993;
   DATA[254,31] := 1.296529;
   DATA[254,32] := 0.7357808;
   DATA[254,33] := 0.306761;
   DATA[254,34] := 2.0;
   DATA[254,35] := 250.8972;
   DATA[254,36] := 1.649953;
   DATA[254,37] := 189.6629;
   DATA[254,38] := 0.000128152;
   DATA[254,39] := 1.0;
   DATA[255,0] := 2.470614;
   DATA[255,1] := 528.5384;
   DATA[255,2] := 2.0;
   DATA[255,3] := 2.0;
   DATA[255,4] := 262.0802;
   DATA[255,5] := 8.39131;
   DATA[255,6] := 328.3517;
   DATA[255,7] := 2.444366;
   DATA[255,8] := 2.0;
   DATA[255,9] := 2.0;
   DATA[255,10] := 2.0;
   DATA[255,11] := 19.72598;
   DATA[255,12] := 2.210678;
   DATA[255,13] := 968.0611;
   DATA[255,14] := 1.0;
   DATA[255,15] := 2.0;
   DATA[255,16] := 1.0;
   DATA[255,17] := 1.0;
   DATA[255,18] := 1.0;
   DATA[255,19] := 2.0;
   DATA[255,20] := 148.808;
   DATA[255,21] := 155.9087;
   DATA[255,22] := 1.718387;
   DATA[255,23] := 962.7147;
   DATA[255,24] := 2.0;
   DATA[255,25] := 2.0;
   DATA[255,26] := 7.876058;
   DATA[255,27] := 144.9885;
   DATA[255,28] := 264.0989;
   DATA[255,29] := 12.15073;
   DATA[255,30] := 1.726993;
   DATA[255,31] := 1.274241;
   DATA[255,32] := 0.7357808;
   DATA[255,33] := 0.306761;
   DATA[255,34] := 2.0;
   DATA[255,35] := 250.8972;
   DATA[255,36] := 1.649953;
   DATA[255,37] := 189.6629;
   DATA[255,38] := 0.000128152;
   DATA[255,39] := 1.0;
   DATA[256,0] := 2.450437;
   DATA[256,1] := 528.1851;
   DATA[256,2] := 2.0;
   DATA[256,3] := 2.0;
   DATA[256,4] := 262.0802;
   DATA[256,5] := 8.393232;
   DATA[256,6] := 328.3517;
   DATA[256,7] := 2.444366;
   DATA[256,8] := 2.0;
   DATA[256,9] := 2.0;
   DATA[256,10] := 2.0;
   DATA[256,11] := 19.72598;
   DATA[256,12] := 2.210678;
   DATA[256,13] := 968.3815;
   DATA[256,14] := 1.0;
   DATA[256,15] := 2.0;
   DATA[256,16] := 1.0;
   DATA[256,17] := 1.0;
   DATA[256,18] := 1.0;
   DATA[256,19] := 2.0;
   DATA[256,20] := 148.808;
   DATA[256,21] := 155.9087;
   DATA[256,22] := 1.718387;
   DATA[256,23] := 962.8685;
   DATA[256,24] := 2.0;
   DATA[256,25] := 2.0;
   DATA[256,26] := 7.876058;
   DATA[256,27] := 144.9885;
   DATA[256,28] := 264.0989;
   DATA[256,29] := 12.15073;
   DATA[256,30] := 1.726993;
   DATA[256,31] := 1.262585;
   DATA[256,32] := 0.7366771;
   DATA[256,33] := 0.306761;
   DATA[256,34] := 2.0;
   DATA[256,35] := 250.8972;
   DATA[256,36] := 1.649953;
   DATA[256,37] := 189.6629;
   DATA[256,38] := 0.000128152;
   DATA[256,39] := 1.0;
   DATA[257,0] := 2.435384;
   DATA[257,1] := 527.6356;
   DATA[257,2] := 2.0;
   DATA[257,3] := 2.0;
   DATA[257,4] := 262.0802;
   DATA[257,5] := 8.393553;
   DATA[257,6] := 328.3517;
   DATA[257,7] := 2.444623;
   DATA[257,8] := 2.0;
   DATA[257,9] := 2.0;
   DATA[257,10] := 2.0;
   DATA[257,11] := 19.73558;
   DATA[257,12] := 2.210678;
   DATA[257,13] := 968.6619;
   DATA[257,14] := 1.0;
   DATA[257,15] := 2.0;
   DATA[257,16] := 1.0;
   DATA[257,17] := 1.0;
   DATA[257,18] := 1.0;
   DATA[257,19] := 2.0;
   DATA[257,20] := 148.808;
   DATA[257,21] := 155.9087;
   DATA[257,22] := 1.718387;
   DATA[257,23] := 963.0223;
   DATA[257,24] := 2.0;
   DATA[257,25] := 2.0;
   DATA[257,26] := 7.876058;
   DATA[257,27] := 144.9885;
   DATA[257,28] := 264.0989;
   DATA[257,29] := 12.15073;
   DATA[257,30] := 1.726993;
   DATA[257,31] := 1.254515;
   DATA[257,32] := 0.7366771;
   DATA[257,33] := 0.306761;
   DATA[257,34] := 2.0;
   DATA[257,35] := 250.8972;
   DATA[257,36] := 1.649953;
   DATA[257,37] := 189.6629;
   DATA[257,38] := 0.000128152;
   DATA[257,39] := 1.0;
   DATA[258,0] := 2.43058;
   DATA[258,1] := 527.6748;
   DATA[258,2] := 2.0;
   DATA[258,3] := 2.0;
   DATA[258,4] := 262.0802;
   DATA[258,5] := 8.393873;
   DATA[258,6] := 328.3517;
   DATA[258,7] := 2.444623;
   DATA[258,8] := 2.0;
   DATA[258,9] := 2.0;
   DATA[258,10] := 2.0;
   DATA[258,11] := 19.70997;
   DATA[258,12] := 2.210678;
   DATA[258,13] := 968.4216;
   DATA[258,14] := 1.0;
   DATA[258,15] := 2.0;
   DATA[258,16] := 1.0;
   DATA[258,17] := 1.0;
   DATA[258,18] := 1.0;
   DATA[258,19] := 2.0;
   DATA[258,20] := 148.808;
   DATA[258,21] := 155.9087;
   DATA[258,22] := 1.718387;
   DATA[258,23] := 963.0223;
   DATA[258,24] := 2.0;
   DATA[258,25] := 2.0;
   DATA[258,26] := 7.876058;
   DATA[258,27] := 144.9885;
   DATA[258,28] := 264.0989;
   DATA[258,29] := 12.15073;
   DATA[258,30] := 1.728916;
   DATA[258,31] := 1.257589;
   DATA[258,32] := 0.7360369;
   DATA[258,33] := 0.306761;
   DATA[258,34] := 2.0;
   DATA[258,35] := 251.0414;
   DATA[258,36] := 1.649953;
   DATA[258,37] := 189.6949;
   DATA[258,38] := 0.000128152;
   DATA[258,39] := 1.0;
   DATA[259,0] := 2.43058;
   DATA[259,1] := 527.8711;
   DATA[259,2] := 2.0;
   DATA[259,3] := 2.0;
   DATA[259,4] := 262.0802;
   DATA[259,5] := 8.393873;
   DATA[259,6] := 328.3517;
   DATA[259,7] := 2.444623;
   DATA[259,8] := 2.0;
   DATA[259,9] := 2.0;
   DATA[259,10] := 2.0;
   DATA[259,11] := 19.64594;
   DATA[259,12] := 2.210678;
   DATA[259,13] := 968.1412;
   DATA[259,14] := 1.0;
   DATA[259,15] := 2.0;
   DATA[259,16] := 1.0;
   DATA[259,17] := 1.0;
   DATA[259,18] := 1.0;
   DATA[259,19] := 2.0;
   DATA[259,20] := 148.808;
   DATA[259,21] := 155.9087;
   DATA[259,22] := 1.718387;
   DATA[259,23] := 963.4068;
   DATA[259,24] := 2.0;
   DATA[259,25] := 2.0;
   DATA[259,26] := 7.876058;
   DATA[259,27] := 144.9885;
   DATA[259,28] := 264.0989;
   DATA[259,29] := 12.15073;
   DATA[259,30] := 1.7293;
   DATA[259,31] := 1.261432;
   DATA[259,32] := 0.7351407;
   DATA[259,33] := 0.306761;
   DATA[259,34] := 2.0;
   DATA[259,35] := 251.0414;
   DATA[259,36] := 1.649953;
   DATA[259,37] := 189.8231;
   DATA[259,38] := 0.000128152;
   DATA[259,39] := 1.0;
   DATA[260,0] := 2.458444;
   DATA[260,1] := 527.9496;
   DATA[260,2] := 2.0;
   DATA[260,3] := 2.0;
   DATA[260,4] := 262.0802;
   DATA[260,5] := 8.393873;
   DATA[260,6] := 328.3517;
   DATA[260,7] := 2.444623;
   DATA[260,8] := 2.0;
   DATA[260,9] := 2.0;
   DATA[260,10] := 2.0;
   DATA[260,11] := 19.62033;
   DATA[260,12] := 2.212087;
   DATA[260,13] := 967.8608;
   DATA[260,14] := 1.0;
   DATA[260,15] := 2.0;
   DATA[260,16] := 1.0;
   DATA[260,17] := 1.0;
   DATA[260,18] := 1.0;
   DATA[260,19] := 2.0;
   DATA[260,20] := 148.808;
   DATA[260,21] := 155.9087;
   DATA[260,22] := 1.718387;
   DATA[260,23] := 962.9838;
   DATA[260,24] := 2.0;
   DATA[260,25] := 2.0;
   DATA[260,26] := 7.876058;
   DATA[260,27] := 144.9885;
   DATA[260,28] := 264.0989;
   DATA[260,29] := 12.15073;
   DATA[260,30] := 1.7293;
   DATA[260,31] := 1.261432;
   DATA[260,32] := 0.7351407;
   DATA[260,33] := 0.306761;
   DATA[260,34] := 2.0;
   DATA[260,35] := 251.0414;
   DATA[260,36] := 1.649953;
   DATA[260,37] := 189.8231;
   DATA[260,38] := 0.000128152;
   DATA[260,39] := 1.0;
   DATA[261,0] := 2.501681;
   DATA[261,1] := 527.5571;
   DATA[261,2] := 2.0;
   DATA[261,3] := 2.0;
   DATA[261,4] := 262.0802;
   DATA[261,5] := 8.393873;
   DATA[261,6] := 328.3517;
   DATA[261,7] := 2.444623;
   DATA[261,8] := 2.0;
   DATA[261,9] := 2.0;
   DATA[261,10] := 2.0;
   DATA[261,11] := 19.62033;
   DATA[261,12] := 2.212984;
   DATA[261,13] := 968.3415;
   DATA[261,14] := 1.0;
   DATA[261,15] := 2.0;
   DATA[261,16] := 1.0;
   DATA[261,17] := 1.0;
   DATA[261,18] := 1.0;
   DATA[261,19] := 2.0;
   DATA[261,20] := 148.808;
   DATA[261,21] := 155.9087;
   DATA[261,22] := 1.718643;
   DATA[261,23] := 962.9838;
   DATA[261,24] := 2.0;
   DATA[261,25] := 2.0;
   DATA[261,26] := 7.876058;
   DATA[261,27] := 144.9885;
   DATA[261,28] := 264.0989;
   DATA[261,29] := 12.15073;
